Yaskawa INFORM job: A_ROOF_SIDE_0617_2_PAINT_14.JBI

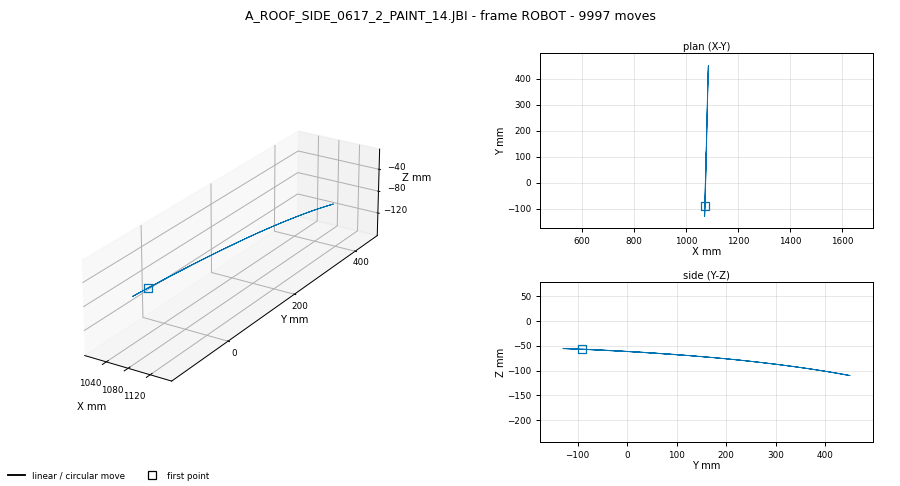
[picture p0: tool path of A_ROOF_SIDE_0617_2_PAINT_14.JBI in frame ROBOT, 9997 of 9997 moves have a stored position in this frame; points joined in program order, loops and branches not executed]
/JOB
//NAME A_ROOF_SIDE_0617_2_PAINT14
//POS
///NPOS 9997,0,0,0,0,0
///TOOL 1
///USER 0
///POSTYPE ROBOT
///RECTAN
///RCONF 1,0,0,0,0,0,0,0,0,0,0,0,0,0,0,0,0,0,0,0,0,0,0,0
C00000=1074.088,-91.546,-56.460,172.902,21.218,153.796
C00001=1074.095,-91.297,-56.470,172.904,21.219,153.796
C00002=1074.101,-91.048,-56.481,172.905,21.220,153.796
C00003=1074.107,-90.797,-56.491,172.907,21.222,153.796
C00004=1074.113,-90.548,-56.502,172.908,21.223,153.796
C00005=1074.120,-90.298,-56.512,172.910,21.225,153.796
C00006=1074.125,-90.048,-56.522,172.911,21.226,153.796
C00007=1074.131,-89.799,-56.533,172.913,21.228,153.796
C00008=1074.138,-89.549,-56.544,172.914,21.229,153.796
C00009=1074.143,-89.299,-56.554,172.916,21.231,153.796
C00010=1074.150,-89.050,-56.564,172.917,21.232,153.796
C00011=1074.156,-88.800,-56.575,172.919,21.234,153.796
C00012=1074.161,-88.550,-56.585,172.921,21.235,153.796
C00013=1074.168,-88.300,-56.596,172.922,21.237,153.796
C00014=1074.174,-88.051,-56.607,172.924,21.238,153.796
C00015=1074.180,-87.801,-56.617,172.925,21.239,153.796
C00016=1074.186,-87.551,-56.627,172.927,21.241,153.797
C00017=1074.192,-87.301,-56.639,172.928,21.242,153.797
C00018=1074.198,-87.052,-56.649,172.930,21.244,153.797
C00019=1074.204,-86.803,-56.660,172.931,21.246,153.797
C00020=1074.210,-86.552,-56.670,172.933,21.247,153.797
C00021=1074.217,-86.303,-56.681,172.934,21.248,153.797
C00022=1074.222,-86.053,-56.692,172.936,21.250,153.797
C00023=1074.229,-85.804,-56.702,172.937,21.251,153.797
C00024=1074.235,-85.554,-56.713,172.939,21.253,153.797
C00025=1074.241,-85.304,-56.723,172.941,21.254,153.797
C00026=1074.247,-85.054,-56.734,172.942,21.255,153.797
C00027=1074.253,-84.805,-56.744,172.943,21.257,153.797
C00028=1074.259,-84.555,-56.756,172.945,21.259,153.797
C00029=1074.266,-84.306,-56.766,172.947,21.260,153.797
C00030=1074.271,-84.055,-56.776,172.948,21.262,153.797
C00031=1074.277,-83.806,-56.787,172.950,21.263,153.797
C00032=1074.284,-83.556,-56.798,172.951,21.264,153.797
C00033=1074.290,-83.307,-56.808,172.953,21.266,153.797
C00034=1074.296,-83.057,-56.819,172.954,21.268,153.797
C00035=1074.303,-82.807,-56.830,172.956,21.269,153.797
C00036=1074.308,-82.558,-56.841,172.957,21.271,153.797
C00037=1074.314,-82.308,-56.851,172.959,21.272,153.797
C00038=1074.321,-82.029,-56.863,172.961,21.274,153.797
C00039=1074.328,-81.750,-56.875,172.962,21.276,153.797
C00040=1074.335,-81.471,-56.887,172.964,21.277,153.797
C00041=1074.342,-81.192,-56.899,172.965,21.279,153.798
C00042=1074.348,-80.942,-56.910,172.967,21.281,153.798
C00043=1074.354,-80.693,-56.921,172.968,21.282,153.798
C00044=1074.361,-80.443,-56.932,172.971,21.284,153.798
C00045=1074.366,-80.193,-56.943,172.972,21.285,153.798
C00046=1074.372,-79.944,-56.953,172.974,21.287,153.798
C00047=1074.379,-79.694,-56.964,172.975,21.289,153.798
C00048=1074.385,-79.444,-56.975,172.977,21.290,153.798
C00049=1074.391,-79.195,-56.986,172.978,21.292,153.798
C00050=1074.397,-78.945,-56.997,172.980,21.294,153.798
C00051=1074.403,-78.695,-57.008,172.981,21.295,153.798
C00052=1074.409,-78.446,-57.019,172.983,21.297,153.798
C00053=1074.415,-78.196,-57.030,172.984,21.298,153.798
C00054=1074.421,-77.946,-57.041,172.986,21.300,153.798
C00055=1074.426,-77.697,-57.052,172.987,21.302,153.798
C00056=1074.434,-77.447,-57.062,172.989,21.303,153.798
C00057=1074.439,-77.197,-57.073,172.990,21.305,153.799
C00058=1074.445,-76.948,-57.084,172.992,21.306,153.799
C00059=1074.451,-76.698,-57.095,172.993,21.308,153.799
C00060=1074.457,-76.448,-57.106,172.995,21.310,153.799
C00061=1074.463,-76.199,-57.117,172.996,21.311,153.799
C00062=1074.469,-75.948,-57.128,172.997,21.313,153.799
C00063=1074.475,-75.699,-57.139,172.999,21.315,153.799
C00064=1074.481,-75.449,-57.150,173.001,21.316,153.799
C00065=1074.487,-75.199,-57.161,173.002,21.318,153.799
C00066=1074.493,-74.950,-57.172,173.003,21.319,153.799
C00067=1074.500,-74.700,-57.183,173.005,21.321,153.799
C00068=1074.506,-74.450,-57.194,173.006,21.323,153.799
C00069=1074.512,-74.201,-57.205,173.008,21.324,153.799
C00070=1074.518,-73.951,-57.217,173.009,21.326,153.800
C00071=1074.524,-73.702,-57.228,173.011,21.328,153.800
C00072=1074.529,-73.452,-57.238,173.012,21.329,153.800
C00073=1074.535,-73.202,-57.250,173.014,21.331,153.800
C00074=1074.541,-72.952,-57.261,173.015,21.333,153.800
C00075=1074.547,-72.702,-57.272,173.016,21.335,153.800
C00076=1074.553,-72.453,-57.283,173.019,21.337,153.800
C00077=1074.559,-72.204,-57.295,173.020,21.339,153.800
C00078=1074.565,-71.954,-57.306,173.022,21.340,153.800
C00079=1074.571,-71.704,-57.317,173.023,21.342,153.800
C00080=1074.577,-71.455,-57.328,173.025,21.343,153.800
C00081=1074.582,-71.204,-57.340,173.026,21.345,153.800
C00082=1074.588,-70.955,-57.351,173.027,21.347,153.801
C00083=1074.594,-70.706,-57.362,173.029,21.349,153.801
C00084=1074.600,-70.456,-57.373,173.030,21.351,153.801
C00085=1074.606,-70.206,-57.384,173.032,21.352,153.801
C00086=1074.612,-69.956,-57.396,173.033,21.354,153.801
C00087=1074.619,-69.707,-57.407,173.035,21.356,153.801
C00088=1074.624,-69.457,-57.419,173.036,21.357,153.801
C00089=1074.630,-69.207,-57.430,173.037,21.359,153.801
C00090=1074.636,-68.957,-57.441,173.039,21.361,153.801
C00091=1074.642,-68.708,-57.453,173.040,21.363,153.802
C00092=1074.648,-68.458,-57.464,173.042,21.365,153.802
C00093=1074.654,-68.209,-57.474,173.043,21.366,153.802
C00094=1074.660,-67.959,-57.487,173.045,21.368,153.802
C00095=1074.665,-67.710,-57.498,173.046,21.370,153.802
C00096=1074.672,-67.459,-57.509,173.048,21.372,153.802
C00097=1074.677,-67.210,-57.520,173.050,21.374,153.802
C00098=1074.684,-66.960,-57.532,173.051,21.376,153.802
C00099=1074.690,-66.711,-57.543,173.053,21.377,153.802
C00100=1074.695,-66.460,-57.555,173.054,21.379,153.802
C00101=1074.701,-66.211,-57.566,173.055,21.381,153.803
C00102=1074.708,-65.934,-57.579,173.057,21.383,153.803
C00103=1074.715,-65.658,-57.592,173.058,21.384,153.803
C00104=1074.721,-65.381,-57.604,173.060,21.387,153.803
C00105=1074.728,-65.104,-57.616,173.062,21.389,153.803
C00106=1074.734,-64.855,-57.628,173.063,21.391,153.803
C00107=1074.740,-64.605,-57.639,173.065,21.392,153.803
C00108=1074.747,-64.356,-57.651,173.066,21.394,153.803
C00109=1074.752,-64.106,-57.662,173.067,21.396,153.804
C00110=1074.758,-63.856,-57.674,173.069,21.397,153.804
C00111=1074.764,-63.607,-57.685,173.070,21.399,153.804
C00112=1074.770,-63.357,-57.697,173.072,21.401,153.804
C00113=1074.776,-63.107,-57.709,173.073,21.403,153.804
C00114=1074.782,-62.857,-57.720,173.075,21.405,153.804
C00115=1074.788,-62.608,-57.732,173.077,21.407,153.804
C00116=1074.794,-62.358,-57.743,173.078,21.409,153.804
C00117=1074.800,-62.109,-57.754,173.080,21.410,153.804
C00118=1074.806,-61.859,-57.766,173.081,21.412,153.804
C00119=1074.812,-61.609,-57.777,173.082,21.414,153.805
C00120=1074.818,-61.360,-57.789,173.084,21.416,153.805
C00121=1074.825,-61.109,-57.800,173.085,21.418,153.805
C00122=1074.830,-60.860,-57.813,173.087,21.420,153.805
C00123=1074.836,-60.610,-57.824,173.088,21.422,153.805
C00124=1074.842,-60.361,-57.835,173.090,21.423,153.805
C00125=1074.849,-60.111,-57.847,173.091,21.425,153.805
C00126=1074.854,-59.862,-57.859,173.092,21.427,153.805
C00127=1074.860,-59.612,-57.870,173.094,21.429,153.806
C00128=1074.867,-59.362,-57.882,173.095,21.430,153.806
C00129=1074.872,-59.112,-57.893,173.097,21.433,153.806
C00130=1074.879,-58.863,-57.905,173.099,21.435,153.806
C00131=1074.884,-58.613,-57.916,173.100,21.437,153.806
C00132=1074.891,-58.364,-57.928,173.102,21.438,153.806
C00133=1074.897,-58.114,-57.941,173.103,21.440,153.806
C00134=1074.903,-57.864,-57.952,173.104,21.442,153.806
C00135=1074.909,-57.615,-57.964,173.106,21.444,153.807
C00136=1074.914,-57.365,-57.975,173.107,21.446,153.807
C00137=1074.921,-57.115,-57.987,173.109,21.447,153.807
C00138=1074.928,-56.866,-57.999,173.110,21.449,153.807
C00139=1074.933,-56.616,-58.010,173.111,21.451,153.807
C00140=1074.939,-56.366,-58.022,173.113,21.453,153.807
C00141=1074.946,-56.116,-58.034,173.114,21.455,153.807
C00142=1074.952,-55.867,-58.045,173.117,21.457,153.807
C00143=1074.958,-55.617,-58.058,173.118,21.459,153.807
C00144=1074.964,-55.367,-58.069,173.119,21.461,153.808
C00145=1074.970,-55.118,-58.081,173.121,21.463,153.808
C00146=1074.976,-54.869,-58.093,173.122,21.465,153.808
C00147=1074.982,-54.618,-58.104,173.124,21.466,153.808
C00148=1074.988,-54.369,-58.116,173.125,21.468,153.808
C00149=1074.994,-54.120,-58.129,173.126,21.470,153.808
C00150=1075.001,-53.869,-58.140,173.128,21.472,153.808
C00151=1075.007,-53.621,-58.151,173.129,21.474,153.809
C00152=1075.013,-53.371,-58.164,173.130,21.476,153.809
C00153=1075.019,-53.120,-58.175,173.132,21.477,153.809
C00154=1075.025,-52.872,-58.187,173.134,21.480,153.809
C00155=1075.031,-52.622,-58.199,173.135,21.482,153.809
C00156=1075.037,-52.372,-58.211,173.137,21.484,153.809
C00157=1075.043,-52.123,-58.222,173.138,21.486,153.809
C00158=1075.049,-51.873,-58.235,173.140,21.487,153.810
C00159=1075.056,-51.623,-58.247,173.141,21.489,153.810
C00160=1075.062,-51.374,-58.259,173.142,21.491,153.810
C00161=1075.067,-51.124,-58.270,173.144,21.493,153.810
C00162=1075.074,-50.874,-58.282,173.145,21.495,153.810
C00163=1075.080,-50.624,-58.295,173.147,21.497,153.810
C00164=1075.087,-50.375,-58.307,173.148,21.499,153.810
C00165=1075.092,-50.126,-58.319,173.150,21.501,153.810
C00166=1075.098,-49.850,-58.332,173.152,21.503,153.811
C00167=1075.105,-49.574,-58.345,173.153,21.505,153.811
C00168=1075.112,-49.299,-58.359,173.154,21.507,153.811
C00169=1075.118,-49.023,-58.372,173.156,21.510,153.811
C00170=1075.124,-48.774,-58.383,173.158,21.512,153.811
C00171=1075.130,-48.524,-58.396,173.159,21.514,153.811
C00172=1075.136,-48.274,-58.408,173.160,21.516,153.812
C00173=1075.142,-48.025,-58.420,173.162,21.518,153.812
C00174=1075.148,-47.776,-58.432,173.163,21.520,153.812
C00175=1075.154,-47.525,-58.444,173.164,21.521,153.812
C00176=1075.160,-47.276,-58.456,173.166,21.523,153.812
C00177=1075.166,-47.026,-58.468,173.168,21.526,153.812
C00178=1075.172,-46.777,-58.480,173.169,21.528,153.812
C00179=1075.178,-46.527,-58.493,173.171,21.530,153.813
C00180=1075.184,-46.278,-58.505,173.172,21.532,153.813
C00181=1075.190,-46.028,-58.517,173.173,21.534,153.813
C00182=1075.196,-45.778,-58.530,173.175,21.536,153.813
C00183=1075.201,-45.529,-58.542,173.176,21.537,153.813
C00184=1075.208,-45.279,-58.554,173.178,21.539,153.813
C00185=1075.214,-45.030,-58.566,173.179,21.542,153.814
C00186=1075.220,-44.780,-58.579,173.181,21.544,153.814
C00187=1075.226,-44.530,-58.590,173.182,21.546,153.814
C00188=1075.232,-44.280,-58.602,173.184,21.548,153.814
C00189=1075.237,-44.030,-58.615,173.185,21.550,153.814
C00190=1075.244,-43.781,-58.627,173.186,21.552,153.814
C00191=1075.249,-43.532,-58.639,173.188,21.554,153.815
C00192=1075.255,-43.282,-58.652,173.189,21.556,153.815
C00193=1075.262,-43.032,-58.664,173.190,21.558,153.815
C00194=1075.268,-42.782,-58.676,173.192,21.560,153.815
C00195=1075.273,-42.533,-58.688,173.193,21.562,153.815
C00196=1075.279,-42.283,-58.701,173.195,21.565,153.815
C00197=1075.286,-42.034,-58.713,173.197,21.567,153.816
C00198=1075.292,-41.784,-58.725,173.198,21.569,153.816
C00199=1075.298,-41.535,-58.739,173.199,21.571,153.816
C00200=1075.304,-41.286,-58.750,173.201,21.573,153.816
C00201=1075.310,-41.036,-58.763,173.202,21.574,153.816
C00202=1075.316,-40.786,-58.775,173.203,21.576,153.816
C00203=1075.322,-40.536,-58.788,173.205,21.578,153.817
C00204=1075.328,-40.286,-58.800,173.206,21.580,153.817
C00205=1075.334,-40.037,-58.812,173.208,21.583,153.817
C00206=1075.340,-39.787,-58.825,173.209,21.585,153.817
C00207=1075.346,-39.538,-58.837,173.211,21.587,153.817
C00208=1075.352,-39.288,-58.849,173.212,21.589,153.817
C00209=1075.358,-39.038,-58.862,173.214,21.591,153.818
C00210=1075.364,-38.789,-58.875,173.215,21.593,153.818
C00211=1075.371,-38.539,-58.887,173.216,21.595,153.818
C00212=1075.376,-38.290,-58.899,173.217,21.597,153.818
C00213=1075.382,-38.040,-58.912,173.219,21.599,153.818
C00214=1075.388,-37.790,-58.924,173.221,21.602,153.818
C00215=1075.394,-37.540,-58.937,173.222,21.604,153.819
C00216=1075.400,-37.291,-58.949,173.224,21.606,153.819
C00217=1075.405,-37.042,-58.962,173.225,21.608,153.819
C00218=1075.411,-36.792,-58.975,173.226,21.610,153.819
C00219=1075.417,-36.542,-58.987,173.228,21.612,153.819
C00220=1075.423,-36.292,-59.000,173.229,21.614,153.820
C00221=1075.429,-36.042,-59.012,173.230,21.616,153.820
C00222=1075.435,-35.794,-59.025,173.232,21.619,153.820
C00223=1075.441,-35.544,-59.037,173.234,21.621,153.820
C00224=1075.447,-35.294,-59.050,173.235,21.623,153.820
C00225=1075.453,-35.045,-59.062,173.236,21.625,153.821
C00226=1075.459,-34.795,-59.075,173.238,21.627,153.821
C00227=1075.465,-34.545,-59.088,173.239,21.629,153.821
C00228=1075.471,-34.295,-59.101,173.240,21.632,153.821
C00229=1075.476,-34.046,-59.113,173.242,21.633,153.821
C00230=1075.484,-33.772,-59.127,173.244,21.636,153.821
C00231=1075.490,-33.496,-59.141,173.245,21.638,153.822
C00232=1075.497,-33.221,-59.156,173.246,21.640,153.822
C00233=1075.503,-32.946,-59.169,173.248,21.643,153.822
C00234=1075.509,-32.696,-59.182,173.250,21.645,153.822
C00235=1075.515,-32.447,-59.195,173.251,21.648,153.823
C00236=1075.521,-32.198,-59.207,173.252,21.650,153.823
C00237=1075.527,-31.948,-59.220,173.254,21.651,153.823
C00238=1075.533,-31.698,-59.233,173.255,21.653,153.823
C00239=1075.539,-31.449,-59.246,173.257,21.656,153.823
C00240=1075.545,-31.199,-59.258,173.258,21.658,153.823
C00241=1075.551,-30.949,-59.271,173.260,21.660,153.824
C00242=1075.557,-30.699,-59.284,173.261,21.663,153.824
C00243=1075.563,-30.450,-59.297,173.262,21.665,153.824
C00244=1075.569,-30.200,-59.310,173.264,21.667,153.824
C00245=1075.575,-29.950,-59.322,173.265,21.669,153.825
C00246=1075.581,-29.701,-59.335,173.266,21.671,153.825
C00247=1075.587,-29.451,-59.348,173.269,21.673,153.825
C00248=1075.593,-29.201,-59.361,173.270,21.675,153.825
C00249=1075.599,-28.952,-59.374,173.271,21.678,153.825
C00250=1075.605,-28.702,-59.387,173.272,21.680,153.825
C00251=1075.611,-28.453,-59.400,173.274,21.682,153.826
C00252=1075.617,-28.204,-59.412,173.275,21.684,153.826
C00253=1075.622,-27.954,-59.425,173.276,21.686,153.826
C00254=1075.629,-27.705,-59.438,173.278,21.688,153.826
C00255=1075.635,-27.455,-59.450,173.280,21.691,153.826
C00256=1075.641,-27.206,-59.464,173.281,21.693,153.827
C00257=1075.647,-26.956,-59.476,173.282,21.695,153.827
C00258=1075.653,-26.706,-59.489,173.284,21.697,153.827
C00259=1075.658,-26.456,-59.503,173.285,21.699,153.827
C00260=1075.664,-26.207,-59.516,173.286,21.702,153.827
C00261=1075.670,-25.957,-59.528,173.288,21.704,153.828
C00262=1075.676,-25.708,-59.542,173.290,21.706,153.828
C00263=1075.682,-25.458,-59.554,173.291,21.709,153.828
C00264=1075.688,-25.208,-59.568,173.292,21.710,153.828
C00265=1075.694,-24.958,-59.581,173.294,21.713,153.828
C00266=1075.700,-24.709,-59.594,173.295,21.715,153.829
C00267=1075.706,-24.459,-59.607,173.296,21.717,153.829
C00268=1075.712,-24.210,-59.620,173.297,21.719,153.829
C00269=1075.718,-23.960,-59.634,173.300,21.722,153.829
C00270=1075.723,-23.711,-59.646,173.301,21.724,153.830
C00271=1075.730,-23.461,-59.659,173.302,21.726,153.830
C00272=1075.736,-23.211,-59.672,173.303,21.729,153.830
C00273=1075.741,-22.962,-59.686,173.305,21.730,153.830
C00274=1075.747,-22.712,-59.698,173.306,21.733,153.830
C00275=1075.753,-22.463,-59.712,173.307,21.735,153.831
C00276=1075.759,-22.213,-59.725,173.308,21.737,153.831
C00277=1075.765,-21.963,-59.738,173.311,21.740,153.831
C00278=1075.771,-21.714,-59.751,173.312,21.742,153.831
C00279=1075.777,-21.465,-59.765,173.313,21.744,153.831
C00280=1075.783,-21.215,-59.777,173.315,21.746,153.832
C00281=1075.788,-20.965,-59.791,173.316,21.749,153.832
C00282=1075.795,-20.716,-59.804,173.317,21.751,153.832
C00283=1075.800,-20.466,-59.817,173.318,21.753,153.832
C00284=1075.807,-20.217,-59.830,173.321,21.755,153.832
C00285=1075.812,-19.967,-59.844,173.322,21.758,153.833
C00286=1075.818,-19.717,-59.857,173.323,21.760,153.833
C00287=1075.824,-19.468,-59.870,173.324,21.762,153.833
C00288=1075.831,-19.219,-59.883,173.326,21.764,153.833
C00289=1075.836,-18.969,-59.896,173.327,21.767,153.834
C00290=1075.842,-18.719,-59.910,173.328,21.769,153.834
C00291=1075.849,-18.469,-59.923,173.330,21.772,153.834
C00292=1075.854,-18.220,-59.937,173.332,21.773,153.834
C00293=1075.860,-17.970,-59.950,173.333,21.776,153.834
C00294=1075.866,-17.695,-59.964,173.334,21.778,153.835
C00295=1075.873,-17.419,-59.979,173.336,21.781,153.835
C00296=1075.880,-17.143,-59.994,173.337,21.783,153.835
C00297=1075.887,-16.866,-60.009,173.339,21.785,153.835
C00298=1075.893,-16.617,-60.022,173.341,21.788,153.836
C00299=1075.899,-16.368,-60.035,173.342,21.790,153.836
C00300=1075.904,-16.118,-60.048,173.343,21.792,153.836
C00301=1075.910,-15.868,-60.062,173.345,21.794,153.836
C00302=1075.917,-15.619,-60.075,173.346,21.797,153.836
C00303=1075.922,-15.370,-60.089,173.347,21.799,153.837
C00304=1075.928,-15.120,-60.102,173.349,21.801,153.837
C00305=1075.935,-14.870,-60.116,173.351,21.804,153.837
C00306=1075.940,-14.620,-60.129,173.352,21.806,153.837
C00307=1075.947,-14.371,-60.142,173.353,21.809,153.838
C00308=1075.952,-14.121,-60.156,173.354,21.811,153.838
C00309=1075.958,-13.872,-60.169,173.356,21.813,153.838
C00310=1075.964,-13.623,-60.183,173.357,21.815,153.838
C00311=1075.970,-13.373,-60.196,173.359,21.818,153.839
C00312=1075.975,-13.124,-60.210,173.360,21.820,153.839
C00313=1075.981,-12.874,-60.223,173.362,21.822,153.839
C00314=1075.987,-12.624,-60.237,173.363,21.825,153.839
C00315=1075.994,-12.374,-60.250,173.364,21.827,153.839
C00316=1075.999,-12.125,-60.264,173.365,21.829,153.840
C00317=1076.005,-11.875,-60.277,173.367,21.831,153.840
C00318=1076.011,-11.626,-60.291,173.369,21.834,153.840
C00319=1076.016,-11.376,-60.305,173.370,21.836,153.840
C00320=1076.022,-11.127,-60.318,173.371,21.838,153.841
C00321=1076.028,-10.877,-60.332,173.373,21.841,153.841
C00322=1076.035,-10.627,-60.346,173.374,21.843,153.841
C00323=1076.040,-10.378,-60.360,173.375,21.845,153.841
C00324=1076.046,-10.129,-60.373,173.377,21.848,153.842
C00325=1076.052,-9.879,-60.387,173.379,21.850,153.842
C00326=1076.058,-9.630,-60.400,173.380,21.853,153.842
C00327=1076.064,-9.380,-60.414,173.381,21.855,153.842
C00328=1076.070,-9.130,-60.428,173.382,21.857,153.842
C00329=1076.076,-8.881,-60.442,173.383,21.859,153.843
C00330=1076.082,-8.631,-60.455,173.386,21.862,153.843
C00331=1076.088,-8.382,-60.469,173.387,21.864,153.843
C00332=1076.093,-8.132,-60.483,173.388,21.866,153.843
C00333=1076.100,-7.882,-60.496,173.389,21.869,153.844
C00334=1076.105,-7.633,-60.510,173.391,21.871,153.844
C00335=1076.112,-7.383,-60.523,173.392,21.873,153.844
C00336=1076.117,-7.134,-60.537,173.393,21.876,153.844
C00337=1076.123,-6.885,-60.550,173.395,21.878,153.844
C00338=1076.129,-6.634,-60.565,173.397,21.880,153.845
C00339=1076.135,-6.385,-60.579,173.398,21.883,153.845
C00340=1076.141,-6.135,-60.592,173.399,21.885,153.845
C00341=1076.147,-5.887,-60.606,173.400,21.887,153.846
C00342=1076.154,-5.637,-60.620,173.402,21.889,153.846
C00343=1076.159,-5.387,-60.634,173.404,21.892,153.846
C00344=1076.165,-5.137,-60.648,173.405,21.895,153.846
C00345=1076.171,-4.888,-60.661,173.406,21.896,153.846
C00346=1076.177,-4.638,-60.675,173.408,21.899,153.847
C00347=1076.183,-4.389,-60.689,173.409,21.901,153.847
C00348=1076.189,-4.139,-60.702,173.410,21.903,153.847
C00349=1076.195,-3.889,-60.717,173.412,21.906,153.847
C00350=1076.201,-3.640,-60.731,173.414,21.908,153.848
C00351=1076.207,-3.391,-60.745,173.415,21.911,153.848
C00352=1076.212,-3.141,-60.758,173.416,21.913,153.848
C00353=1076.219,-2.891,-60.772,173.417,21.915,153.848
C00354=1076.225,-2.642,-60.787,173.419,21.918,153.849
C00355=1076.230,-2.392,-60.800,173.421,21.920,153.849
C00356=1076.236,-2.143,-60.814,173.422,21.923,153.849
C00357=1076.241,-1.893,-60.828,173.423,21.925,153.849
C00358=1076.248,-1.616,-60.844,173.424,21.927,153.850
C00359=1076.255,-1.338,-60.859,173.426,21.930,153.850
C00360=1076.261,-1.060,-60.875,173.428,21.933,153.850
C00361=1076.268,-0.783,-60.890,173.429,21.936,153.850
C00362=1076.273,-0.534,-60.905,173.431,21.938,153.851
C00363=1076.279,-0.284,-60.919,173.432,21.940,153.851
C00364=1076.285,-0.034,-60.933,173.433,21.943,153.851
C00365=1076.290,0.215,-60.947,173.434,21.945,153.852
C00366=1076.296,0.464,-60.962,173.436,21.947,153.852
C00367=1076.302,0.714,-60.975,173.438,21.950,153.852
C00368=1076.309,0.964,-60.989,173.439,21.953,153.852
C00369=1076.314,1.213,-61.004,173.440,21.955,153.853
C00370=1076.320,1.462,-61.018,173.442,21.957,153.853
C00371=1076.325,1.712,-61.031,173.443,21.960,153.853
C00372=1076.332,1.962,-61.046,173.444,21.962,153.853
C00373=1076.337,2.211,-61.060,173.446,21.964,153.853
C00374=1076.343,2.461,-61.074,173.447,21.967,153.854
C00375=1076.349,2.710,-61.089,173.449,21.969,153.854
C00376=1076.355,2.960,-61.102,173.450,21.972,153.854
C00377=1076.361,3.209,-61.116,173.451,21.974,153.854
C00378=1076.367,3.459,-61.131,173.452,21.976,153.855
C00379=1076.373,3.709,-61.145,173.454,21.979,153.855
C00380=1076.378,3.957,-61.160,173.456,21.981,153.855
C00381=1076.384,4.208,-61.174,173.457,21.983,153.855
C00382=1076.390,4.457,-61.188,173.458,21.986,153.856
C00383=1076.396,4.706,-61.202,173.459,21.988,153.856
C00384=1076.402,4.957,-61.216,173.461,21.991,153.856
C00385=1076.408,5.206,-61.231,173.463,21.993,153.856
C00386=1076.413,5.455,-61.245,173.464,21.996,153.857
C00387=1076.419,5.705,-61.260,173.465,21.998,153.857
C00388=1076.425,5.954,-61.274,173.466,22.001,153.857
C00389=1076.431,6.203,-61.288,173.468,22.002,153.857
C00390=1076.437,6.453,-61.302,173.470,22.005,153.858
C00391=1076.443,6.702,-61.316,173.471,22.008,153.858
C00392=1076.449,6.952,-61.331,173.472,22.010,153.858
C00393=1076.455,7.201,-61.345,173.474,22.012,153.858
C00394=1076.461,7.451,-61.359,173.475,22.015,153.859
C00395=1076.467,7.701,-61.374,173.476,22.017,153.859
C00396=1076.472,7.950,-61.388,173.478,22.020,153.859
C00397=1076.479,8.200,-61.403,173.480,22.022,153.859
C00398=1076.484,8.449,-61.417,173.481,22.024,153.860
C00399=1076.490,8.698,-61.431,173.482,22.027,153.860
C00400=1076.496,8.949,-61.446,173.483,22.029,153.860
C00401=1076.502,9.198,-61.460,173.485,22.032,153.860
C00402=1076.508,9.448,-61.474,173.487,22.034,153.861
C00403=1076.514,9.697,-61.489,173.488,22.037,153.861
C00404=1076.520,9.947,-61.504,173.489,22.039,153.861
C00405=1076.526,10.196,-61.518,173.490,22.041,153.862
C00406=1076.532,10.446,-61.533,173.492,22.043,153.862
C00407=1076.537,10.695,-61.547,173.494,22.046,153.862
C00408=1076.543,10.944,-61.561,173.495,22.048,153.862
C00409=1076.550,11.194,-61.576,173.496,22.051,153.862
C00410=1076.555,11.444,-61.590,173.497,22.053,153.863
C00411=1076.562,11.693,-61.605,173.499,22.056,153.863
C00412=1076.567,11.942,-61.620,173.501,22.058,153.863
C00413=1076.573,12.192,-61.634,173.502,22.060,153.863
C00414=1076.579,12.441,-61.648,173.503,22.063,153.864
C00415=1076.586,12.691,-61.663,173.505,22.065,153.864
C00416=1076.591,12.941,-61.677,173.506,22.067,153.864
C00417=1076.597,13.190,-61.692,173.508,22.070,153.864
C00418=1076.603,13.439,-61.707,173.509,22.073,153.865
C00419=1076.609,13.690,-61.721,173.510,22.075,153.865
C00420=1076.615,13.938,-61.735,173.512,22.077,153.865
C00421=1076.621,14.188,-61.750,173.513,22.079,153.866
C00422=1076.628,14.468,-61.766,173.515,22.082,153.866
C00423=1076.635,14.747,-61.783,173.516,22.085,153.866
C00424=1076.641,15.026,-61.799,173.518,22.088,153.866
C00425=1076.647,15.306,-61.816,173.519,22.090,153.867
C00426=1076.653,15.556,-61.831,173.521,22.093,153.867
C00427=1076.659,15.805,-61.845,173.522,22.095,153.867
C00428=1076.665,16.054,-61.860,173.524,22.098,153.867
C00429=1076.671,16.304,-61.875,173.525,22.100,153.868
C00430=1076.677,16.554,-61.890,173.526,22.102,153.868
C00431=1076.682,16.803,-61.904,173.528,22.105,153.868
C00432=1076.689,17.053,-61.919,173.529,22.107,153.869
C00433=1076.695,17.302,-61.934,173.531,22.110,153.869
C00434=1076.700,17.552,-61.949,173.532,22.113,153.869
C00435=1076.706,17.801,-61.963,173.534,22.114,153.869
C00436=1076.712,18.051,-61.978,173.535,22.117,153.870
C00437=1076.718,18.300,-61.993,173.536,22.119,153.870
C00438=1076.723,18.550,-62.008,173.538,22.122,153.870
C00439=1076.729,18.799,-62.023,173.539,22.125,153.870
C00440=1076.736,19.048,-62.038,173.540,22.127,153.871
C00441=1076.741,19.297,-62.052,173.542,22.129,153.871
C00442=1076.747,19.548,-62.067,173.543,22.132,153.871
C00443=1076.753,19.797,-62.082,173.545,22.134,153.871
C00444=1076.759,20.046,-62.097,173.546,22.137,153.872
C00445=1076.765,20.296,-62.112,173.548,22.139,153.872
C00446=1076.770,20.545,-62.127,173.549,22.141,153.872
C00447=1076.777,20.795,-62.142,173.550,22.144,153.872
C00448=1076.783,21.044,-62.156,173.552,22.147,153.873
C00449=1076.788,21.294,-62.172,173.553,22.149,153.873
C00450=1076.794,21.543,-62.186,173.555,22.151,153.873
C00451=1076.800,21.793,-62.202,173.556,22.154,153.874
C00452=1076.805,22.042,-62.216,173.557,22.156,153.874
C00453=1076.812,22.291,-62.231,173.559,22.159,153.874
C00454=1076.817,22.541,-62.247,173.560,22.161,153.874
C00455=1076.823,22.790,-62.262,173.562,22.164,153.875
C00456=1076.830,23.040,-62.277,173.563,22.166,153.875
C00457=1076.835,23.289,-62.292,173.564,22.169,153.875
C00458=1076.841,23.539,-62.307,173.566,22.171,153.875
C00459=1076.847,23.789,-62.322,173.568,22.173,153.876
C00460=1076.852,24.038,-62.337,173.569,22.176,153.876
C00461=1076.859,24.288,-62.352,173.570,22.178,153.876
C00462=1076.864,24.537,-62.367,173.571,22.181,153.876
C00463=1076.870,24.786,-62.382,173.573,22.184,153.877
C00464=1076.876,25.036,-62.397,173.574,22.186,153.877
C00465=1076.882,25.285,-62.412,173.576,22.188,153.877
C00466=1076.888,25.535,-62.427,173.577,22.190,153.877
C00467=1076.893,25.784,-62.442,173.578,22.193,153.878
C00468=1076.899,26.034,-62.457,173.580,22.196,153.878
C00469=1076.905,26.284,-62.473,173.582,22.198,153.878
C00470=1076.911,26.533,-62.487,173.583,22.200,153.878
C00471=1076.917,26.783,-62.502,173.584,22.202,153.879
C00472=1076.923,27.032,-62.518,173.585,22.205,153.879
C00473=1076.929,27.281,-62.533,173.587,22.208,153.879
C00474=1076.935,27.531,-62.548,173.589,22.210,153.880
C00475=1076.940,27.780,-62.563,173.590,22.213,153.880
C00476=1076.946,28.030,-62.579,173.591,22.215,153.880
C00477=1076.952,28.279,-62.594,173.593,22.218,153.880
C00478=1076.958,28.529,-62.609,173.595,22.220,153.881
C00479=1076.964,28.778,-62.624,173.596,22.222,153.881
C00480=1076.970,29.028,-62.640,173.597,22.225,153.881
C00481=1076.976,29.277,-62.654,173.598,22.227,153.881
C00482=1076.981,29.527,-62.670,173.600,22.230,153.882
C00483=1076.987,29.777,-62.686,173.601,22.233,153.882
C00484=1076.993,30.025,-62.701,173.603,22.235,153.882
C00485=1076.999,30.275,-62.716,173.604,22.237,153.882
C00486=1077.005,30.556,-62.733,173.606,22.240,153.883
C00487=1077.012,30.836,-62.750,173.607,22.243,153.883
C00488=1077.018,31.117,-62.768,173.609,22.246,153.883
C00489=1077.025,31.399,-62.785,173.611,22.248,153.884
C00490=1077.031,31.647,-62.801,173.612,22.251,153.884
C00491=1077.036,31.897,-62.816,173.614,22.253,153.884
C00492=1077.043,32.147,-62.831,173.615,22.256,153.885
C00493=1077.048,32.396,-62.847,173.616,22.258,153.885
C00494=1077.054,32.624,-62.861,173.618,22.260,153.885
C00495=1077.059,32.853,-62.875,173.619,22.263,153.885
C00496=1077.064,33.081,-62.890,173.620,22.265,153.886
C00497=1077.069,33.310,-62.903,173.621,22.267,153.886
C00498=1077.074,33.539,-62.917,173.623,22.270,153.886
C00499=1077.080,33.767,-62.931,173.624,22.272,153.886
C00500=1077.085,33.995,-62.946,173.625,22.274,153.886
C00501=1077.090,34.224,-62.960,173.626,22.276,153.887
C00502=1077.097,34.473,-62.975,173.629,22.279,153.887
C00503=1077.103,34.723,-62.991,173.630,22.281,153.887
C00504=1077.108,34.973,-63.007,173.631,22.284,153.888
C00505=1077.114,35.222,-63.022,173.632,22.286,153.888
C00506=1077.120,35.471,-63.038,173.634,22.289,153.888
C00507=1077.126,35.721,-63.053,173.636,22.291,153.888
C00508=1077.132,35.971,-63.068,173.637,22.294,153.889
C00509=1077.138,36.219,-63.084,173.638,22.296,153.889
C00510=1077.143,36.469,-63.100,173.640,22.298,153.889
C00511=1077.150,36.718,-63.115,173.642,22.301,153.889
C00512=1077.156,36.968,-63.131,173.643,22.303,153.890
C00513=1077.161,37.217,-63.146,173.644,22.306,153.890
C00514=1077.167,37.466,-63.162,173.645,22.308,153.890
C00515=1077.173,37.716,-63.177,173.647,22.311,153.890
C00516=1077.179,37.966,-63.194,173.649,22.313,153.891
C00517=1077.184,38.215,-63.209,173.650,22.316,153.891
C00518=1077.191,38.464,-63.224,173.651,22.318,153.891
C00519=1077.196,38.714,-63.240,173.653,22.321,153.891
C00520=1077.202,38.963,-63.256,173.654,22.323,153.892
C00521=1077.207,39.213,-63.271,173.656,22.326,153.892
C00522=1077.213,39.462,-63.288,173.657,22.328,153.892
C00523=1077.219,39.712,-63.303,173.658,22.331,153.893
C00524=1077.226,39.961,-63.319,173.660,22.333,153.893
C00525=1077.231,40.211,-63.334,173.661,22.336,153.893
C00526=1077.237,40.460,-63.350,173.663,22.338,153.893
C00527=1077.242,40.710,-63.366,173.664,22.340,153.894
C00528=1077.248,40.959,-63.382,173.666,22.343,153.894
C00529=1077.254,41.208,-63.398,173.667,22.346,153.894
C00530=1077.260,41.458,-63.414,173.669,22.348,153.895
C00531=1077.265,41.707,-63.430,173.670,22.350,153.895
C00532=1077.271,41.957,-63.445,173.672,22.353,153.895
C00533=1077.277,42.206,-63.461,173.673,22.356,153.895
C00534=1077.283,42.456,-63.477,173.675,22.358,153.896
C00535=1077.289,42.705,-63.493,173.676,22.360,153.896
C00536=1077.294,42.954,-63.509,173.678,22.363,153.896
C00537=1077.300,43.204,-63.524,173.679,22.365,153.896
C00538=1077.306,43.453,-63.541,173.680,22.368,153.897
C00539=1077.312,43.703,-63.557,173.682,22.370,153.897
C00540=1077.318,43.953,-63.572,173.684,22.373,153.897
C00541=1077.323,44.202,-63.589,173.685,22.376,153.898
C00542=1077.329,44.451,-63.604,173.686,22.378,153.898
C00543=1077.334,44.701,-63.620,173.687,22.380,153.898
C00544=1077.340,44.950,-63.636,173.689,22.383,153.898
C00545=1077.346,45.199,-63.653,173.691,22.386,153.899
C00546=1077.351,45.448,-63.668,173.692,22.388,153.899
C00547=1077.357,45.698,-63.684,173.693,22.390,153.899
C00548=1077.363,45.947,-63.700,173.695,22.393,153.899
C00549=1077.369,46.197,-63.716,173.697,22.395,153.900
C00550=1077.376,46.520,-63.737,173.698,22.399,153.900
C00551=1077.384,46.843,-63.758,173.700,22.402,153.900
C00552=1077.391,47.165,-63.778,173.702,22.406,153.901
C00553=1077.398,47.488,-63.800,173.703,22.409,153.901
C00554=1077.404,47.737,-63.816,173.706,22.411,153.901
C00555=1077.410,47.987,-63.831,173.707,22.413,153.902
C00556=1077.416,48.237,-63.848,173.708,22.416,153.902
C00557=1077.422,48.486,-63.864,173.709,22.418,153.902
C00558=1077.428,48.735,-63.880,173.711,22.421,153.903
C00559=1077.433,48.984,-63.896,173.713,22.423,153.903
C00560=1077.438,49.234,-63.912,173.714,22.426,153.903
C00561=1077.444,49.484,-63.929,173.715,22.428,153.903
C00562=1077.450,49.733,-63.945,173.717,22.431,153.904
C00563=1077.456,49.982,-63.961,173.718,22.434,153.904
C00564=1077.462,50.232,-63.977,173.720,22.436,153.904
C00565=1077.468,50.481,-63.994,173.721,22.438,153.905
C00566=1077.473,50.731,-64.009,173.723,22.441,153.905
C00567=1077.478,50.981,-64.026,173.724,22.443,153.905
C00568=1077.484,51.230,-64.042,173.726,22.446,153.905
C00569=1077.490,51.479,-64.058,173.728,22.448,153.906
C00570=1077.496,51.728,-64.074,173.729,22.451,153.906
C00571=1077.502,51.977,-64.091,173.730,22.453,153.906
C00572=1077.508,52.227,-64.107,173.731,22.456,153.906
C00573=1077.514,52.476,-64.123,173.733,22.459,153.907
C00574=1077.519,52.726,-64.140,173.735,22.461,153.907
C00575=1077.525,52.975,-64.156,173.736,22.463,153.907
C00576=1077.531,53.224,-64.173,173.737,22.465,153.907
C00577=1077.537,53.474,-64.189,173.739,22.468,153.908
C00578=1077.543,53.723,-64.205,173.741,22.471,153.908
C00579=1077.547,53.973,-64.221,173.742,22.473,153.908
C00580=1077.553,54.223,-64.237,173.743,22.476,153.909
C00581=1077.559,54.472,-64.254,173.745,22.478,153.909
C00582=1077.565,54.721,-64.270,173.747,22.480,153.909
C00583=1077.571,54.971,-64.286,173.748,22.483,153.909
C00584=1077.577,55.220,-64.302,173.750,22.486,153.910
C00585=1077.583,55.469,-64.320,173.751,22.488,153.910
C00586=1077.589,55.719,-64.336,173.752,22.490,153.910
C00587=1077.595,55.968,-64.353,173.754,22.493,153.910
C00588=1077.601,56.217,-64.369,173.756,22.495,153.911
C00589=1077.606,56.467,-64.386,173.757,22.498,153.911
C00590=1077.612,56.716,-64.402,173.758,22.500,153.911
C00591=1077.618,56.966,-64.418,173.760,22.503,153.911
C00592=1077.624,57.215,-64.434,173.762,22.505,153.912
C00593=1077.630,57.464,-64.451,173.763,22.508,153.912
C00594=1077.635,57.714,-64.467,173.764,22.510,153.912
C00595=1077.641,57.963,-64.484,173.767,22.513,153.912
C00596=1077.647,58.213,-64.500,173.768,22.515,153.913
C00597=1077.653,58.462,-64.516,173.769,22.517,153.913
C00598=1077.658,58.711,-64.534,173.770,22.520,153.913
C00599=1077.664,58.960,-64.550,173.773,22.522,153.913
C00600=1077.670,59.210,-64.566,173.774,22.525,153.914
C00601=1077.676,59.459,-64.583,173.775,22.527,153.914
C00602=1077.681,59.709,-64.599,173.776,22.529,153.914
C00603=1077.688,59.959,-64.616,173.778,22.532,153.915
C00604=1077.694,60.208,-64.633,173.780,22.534,153.915
C00605=1077.700,60.457,-64.649,173.781,22.537,153.915
C00606=1077.705,60.707,-64.666,173.783,22.539,153.915
C00607=1077.711,60.956,-64.682,173.784,22.542,153.916
C00608=1077.717,61.205,-64.699,173.786,22.544,153.916
C00609=1077.723,61.454,-64.716,173.787,22.546,153.916
C00610=1077.729,61.704,-64.732,173.789,22.549,153.916
C00611=1077.735,61.953,-64.749,173.790,22.551,153.917
C00612=1077.741,62.203,-64.765,173.792,22.554,153.917
C00613=1077.746,62.453,-64.782,173.794,22.556,153.917
C00614=1077.753,62.732,-64.801,173.795,22.559,153.917
C00615=1077.760,63.013,-64.819,173.797,22.561,153.918
C00616=1077.766,63.293,-64.839,173.798,22.564,153.918
C00617=1077.773,63.574,-64.857,173.800,22.567,153.918
C00618=1077.779,63.824,-64.873,173.802,22.569,153.918
C00619=1077.785,64.073,-64.891,173.803,22.572,153.919
C00620=1077.791,64.323,-64.908,173.805,22.574,153.919
C00621=1077.797,64.572,-64.924,173.806,22.577,153.919
C00622=1077.803,64.821,-64.941,173.808,22.579,153.919
C00623=1077.809,65.071,-64.958,173.810,22.582,153.920
C00624=1077.814,65.320,-64.975,173.811,22.584,153.920
C00625=1077.820,65.569,-64.992,173.812,22.586,153.920
C00626=1077.825,65.819,-65.008,173.814,22.589,153.921
C00627=1077.831,66.068,-65.025,173.816,22.592,153.921
C00628=1077.837,66.318,-65.043,173.817,22.594,153.921
C00629=1077.843,66.567,-65.059,173.818,22.596,153.921
C00630=1077.848,66.817,-65.076,173.820,22.599,153.922
C00631=1077.855,67.066,-65.093,173.822,22.601,153.922
C00632=1077.860,67.315,-65.110,173.823,22.604,153.922
C00633=1077.866,67.564,-65.127,173.825,22.606,153.922
C00634=1077.871,67.814,-65.143,173.826,22.608,153.923
C00635=1077.878,68.063,-65.161,173.828,22.611,153.923
C00636=1077.883,68.313,-65.178,173.830,22.614,153.923
C00637=1077.889,68.562,-65.194,173.831,22.616,153.923
C00638=1077.895,68.811,-65.211,173.833,22.618,153.924
C00639=1077.900,69.061,-65.228,173.834,22.620,153.924
C00640=1077.906,69.309,-65.245,173.836,22.623,153.924
C00641=1077.912,69.560,-65.262,173.837,22.626,153.924
C00642=1077.918,69.809,-65.280,173.838,22.628,153.925
C00643=1077.924,70.058,-65.296,173.841,22.630,153.925
C00644=1077.929,70.307,-65.314,173.842,22.633,153.925
C00645=1077.935,70.557,-65.330,173.843,22.635,153.925
C00646=1077.941,70.806,-65.348,173.845,22.638,153.926
C00647=1077.946,71.056,-65.365,173.846,22.641,153.926
C00648=1077.953,71.305,-65.382,173.848,22.643,153.926
C00649=1077.958,71.554,-65.399,173.850,22.645,153.926
C00650=1077.963,71.803,-65.416,173.851,22.648,153.927
C00651=1077.970,72.052,-65.433,173.853,22.650,153.927
C00652=1077.976,72.302,-65.450,173.854,22.653,153.927
C00653=1077.981,72.552,-65.468,173.856,22.655,153.928
C00654=1077.986,72.801,-65.485,173.857,22.657,153.928
C00655=1077.993,73.050,-65.502,173.859,22.660,153.928
C00656=1077.998,73.299,-65.519,173.861,22.662,153.928
C00657=1078.004,73.549,-65.537,173.862,22.665,153.929
C00658=1078.010,73.798,-65.554,173.863,22.667,153.929
C00659=1078.016,74.047,-65.571,173.865,22.670,153.929
C00660=1078.021,74.297,-65.588,173.867,22.672,153.929
C00661=1078.027,74.546,-65.606,173.868,22.674,153.930
C00662=1078.033,74.795,-65.623,173.870,22.677,153.930
C00663=1078.038,75.045,-65.640,173.871,22.679,153.930
C00664=1078.044,75.294,-65.657,173.873,22.682,153.930
C00665=1078.050,75.544,-65.675,173.875,22.684,153.931
C00666=1078.056,75.793,-65.692,173.876,22.687,153.931
C00667=1078.062,76.042,-65.709,173.877,22.689,153.931
C00668=1078.067,76.291,-65.727,173.880,22.692,153.931
C00669=1078.073,76.541,-65.744,173.881,22.694,153.932
C00670=1078.079,76.790,-65.761,173.882,22.696,153.932
C00671=1078.085,77.039,-65.778,173.884,22.699,153.932
C00672=1078.090,77.288,-65.796,173.886,22.701,153.932
C00673=1078.096,77.539,-65.813,173.887,22.704,153.933
C00674=1078.102,77.788,-65.831,173.889,22.706,153.933
C00675=1078.108,78.036,-65.848,173.890,22.709,153.933
C00676=1078.114,78.286,-65.866,173.892,22.711,153.933
C00677=1078.119,78.536,-65.883,173.894,22.714,153.934
C00678=1078.125,78.817,-65.903,173.895,22.716,153.934
C00679=1078.132,79.097,-65.922,173.897,22.719,153.934
C00680=1078.138,79.377,-65.942,173.898,22.721,153.934
C00681=1078.145,79.658,-65.961,173.900,22.725,153.935
C00682=1078.150,79.907,-65.979,173.902,22.726,153.935
C00683=1078.156,80.156,-65.996,173.904,22.729,153.935
C00684=1078.162,80.406,-66.014,173.905,22.732,153.936
C00685=1078.168,80.655,-66.032,173.906,22.734,153.936
C00686=1078.173,80.904,-66.049,173.909,22.737,153.936
C00687=1078.179,81.154,-66.067,173.910,22.739,153.936
C00688=1078.184,81.403,-66.084,173.911,22.741,153.937
C00689=1078.190,81.652,-66.102,173.913,22.744,153.937
C00690=1078.195,81.901,-66.119,173.915,22.746,153.937
C00691=1078.202,82.151,-66.137,173.916,22.749,153.937
C00692=1078.207,82.400,-66.155,173.918,22.751,153.938
C00693=1078.213,82.649,-66.172,173.919,22.754,153.938
C00694=1078.219,82.899,-66.190,173.922,22.756,153.938
C00695=1078.224,83.148,-66.208,173.923,22.759,153.938
C00696=1078.230,83.397,-66.225,173.924,22.761,153.939
C00697=1078.236,83.647,-66.243,173.926,22.764,153.939
C00698=1078.241,83.896,-66.261,173.928,22.766,153.939
C00699=1078.247,84.145,-66.278,173.929,22.768,153.939
C00700=1078.253,84.395,-66.296,173.931,22.771,153.940
C00701=1078.259,84.644,-66.314,173.932,22.773,153.940
C00702=1078.265,84.893,-66.332,173.934,22.775,153.940
C00703=1078.270,85.142,-66.349,173.936,22.778,153.940
C00704=1078.276,85.391,-66.367,173.937,22.780,153.941
C00705=1078.282,85.641,-66.385,173.939,22.783,153.941
C00706=1078.287,85.890,-66.402,173.941,22.785,153.941
C00707=1078.293,86.140,-66.420,173.942,22.787,153.941
C00708=1078.299,86.389,-66.438,173.943,22.790,153.942
C00709=1078.305,86.638,-66.456,173.945,22.793,153.942
C00710=1078.311,86.888,-66.473,173.947,22.794,153.942
C00711=1078.316,87.137,-66.491,173.949,22.797,153.942
C00712=1078.322,87.387,-66.509,173.950,22.800,153.943
C00713=1078.328,87.636,-66.527,173.952,22.802,153.943
C00714=1078.333,87.885,-66.544,173.954,22.804,153.943
C00715=1078.339,88.135,-66.563,173.955,22.807,153.943
C00716=1078.345,88.383,-66.581,173.957,22.809,153.943
C00717=1078.351,88.633,-66.599,173.959,22.811,153.944
C00718=1078.356,88.882,-66.616,173.960,22.814,153.944
C00719=1078.362,89.132,-66.634,173.961,22.816,153.944
C00720=1078.368,89.381,-66.652,173.964,22.819,153.944
C00721=1078.374,89.630,-66.670,173.965,22.821,153.945
C00722=1078.379,89.879,-66.687,173.967,22.823,153.945
C00723=1078.386,90.129,-66.706,173.968,22.826,153.945
C00724=1078.391,90.378,-66.724,173.970,22.828,153.945
C00725=1078.398,90.627,-66.742,173.972,22.830,153.946
C00726=1078.403,90.876,-66.759,173.973,22.833,153.946
C00727=1078.408,91.126,-66.777,173.974,22.835,153.946
C00728=1078.414,91.375,-66.796,173.977,22.837,153.946
C00729=1078.420,91.624,-66.814,173.978,22.840,153.947
C00730=1078.425,91.874,-66.832,173.980,22.843,153.947
C00731=1078.431,92.123,-66.850,173.981,22.845,153.947
C00732=1078.437,92.372,-66.868,173.983,22.847,153.947
C00733=1078.443,92.621,-66.886,173.985,22.850,153.948
C00734=1078.448,92.871,-66.904,173.986,22.852,153.948
C00735=1078.454,93.120,-66.922,173.988,22.854,153.948
C00736=1078.459,93.369,-66.940,173.990,22.857,153.948
C00737=1078.465,93.619,-66.959,173.991,22.859,153.949
C00738=1078.470,93.868,-66.976,173.993,22.862,153.949
C00739=1078.477,94.117,-66.995,173.995,22.864,153.949
C00740=1078.482,94.366,-67.013,173.996,22.866,153.949
C00741=1078.488,94.616,-67.031,173.998,22.869,153.949
C00742=1078.494,94.896,-67.052,173.999,22.871,153.950
C00743=1078.500,95.177,-67.072,174.001,22.874,153.950
C00744=1078.507,95.457,-67.093,174.004,22.877,153.950
C00745=1078.513,95.738,-67.113,174.006,22.880,153.951
C00746=1078.520,95.987,-67.131,174.007,22.882,153.951
C00747=1078.524,96.237,-67.149,174.008,22.884,153.951
C00748=1078.531,96.486,-67.168,174.011,22.887,153.951
C00749=1078.536,96.735,-67.186,174.012,22.889,153.952
C00750=1078.542,96.984,-67.205,174.013,22.891,153.952
C00751=1078.547,97.233,-67.222,174.016,22.894,153.952
C00752=1078.554,97.483,-67.240,174.017,22.896,153.952
C00753=1078.559,97.732,-67.259,174.019,22.899,153.953
C00754=1078.565,97.982,-67.277,174.020,22.901,153.953
C00755=1078.571,98.231,-67.296,174.022,22.903,153.953
C00756=1078.576,98.480,-67.314,174.024,22.905,153.953
C00757=1078.582,98.729,-67.333,174.025,22.908,153.953
C00758=1078.587,98.979,-67.351,174.027,22.911,153.954
C00759=1078.594,99.228,-67.369,174.029,22.913,153.954
C00760=1078.599,99.477,-67.387,174.030,22.915,153.954
C00761=1078.605,99.726,-67.406,174.032,22.917,153.954
C00762=1078.611,99.976,-67.424,174.034,22.920,153.955
C00763=1078.617,100.224,-67.442,174.036,22.922,153.955
C00764=1078.622,100.474,-67.461,174.037,22.924,153.955
C00765=1078.628,100.723,-67.479,174.039,22.927,153.955
C00766=1078.633,100.973,-67.498,174.041,22.929,153.955
C00767=1078.640,101.222,-67.516,174.042,22.931,153.956
C00768=1078.645,101.471,-67.535,174.044,22.934,153.956
C00769=1078.651,101.720,-67.553,174.046,22.936,153.956
C00770=1078.656,101.969,-67.572,174.048,22.939,153.956
C00771=1078.662,102.219,-67.590,174.049,22.941,153.957
C00772=1078.668,102.468,-67.609,174.051,22.943,153.957
C00773=1078.674,102.717,-67.628,174.053,22.946,153.957
C00774=1078.679,102.967,-67.646,174.054,22.948,153.957
C00775=1078.684,103.216,-67.665,174.056,22.951,153.958
C00776=1078.690,103.465,-67.683,174.058,22.953,153.958
C00777=1078.695,103.714,-67.702,174.060,22.955,153.958
C00778=1078.702,103.963,-67.720,174.061,22.958,153.958
C00779=1078.707,104.213,-67.739,174.062,22.960,153.959
C00780=1078.712,104.462,-67.758,174.065,22.962,153.959
C00781=1078.719,104.711,-67.777,174.066,22.965,153.959
C00782=1078.724,104.960,-67.796,174.068,22.967,153.959
C00783=1078.730,105.209,-67.813,174.070,22.970,153.960
C00784=1078.736,105.459,-67.833,174.071,22.972,153.960
C00785=1078.741,105.708,-67.852,174.073,22.974,153.960
C00786=1078.747,105.957,-67.869,174.074,22.977,153.960
C00787=1078.752,106.207,-67.889,174.077,22.979,153.960
C00788=1078.758,106.456,-67.908,174.078,22.981,153.961
C00789=1078.764,106.705,-67.926,174.080,22.984,153.961
C00790=1078.769,106.955,-67.945,174.082,22.986,153.961
C00791=1078.775,107.203,-67.963,174.084,22.989,153.961
C00792=1078.781,107.453,-67.982,174.085,22.991,153.962
C00793=1078.787,107.702,-68.001,174.086,22.993,153.962
C00794=1078.793,107.951,-68.020,174.089,22.995,153.962
C00795=1078.798,108.201,-68.038,174.090,22.998,153.962
C00796=1078.803,108.450,-68.058,174.092,23.000,153.962
C00797=1078.810,108.699,-68.076,174.094,23.002,153.963
C00798=1078.815,108.948,-68.095,174.096,23.005,153.963
C00799=1078.821,109.197,-68.114,174.097,23.007,153.963
C00800=1078.827,109.446,-68.133,174.100,23.009,153.963
C00801=1078.832,109.696,-68.151,174.101,23.012,153.964
C00802=1078.838,109.945,-68.170,174.102,23.014,153.964
C00803=1078.844,110.194,-68.189,174.104,23.016,153.964
C00804=1078.850,110.444,-68.208,174.106,23.018,153.964
C00805=1078.855,110.692,-68.227,174.108,23.021,153.964
C00806=1078.862,110.973,-68.248,174.110,23.024,153.965
C00807=1078.868,111.254,-68.270,174.112,23.026,153.965
C00808=1078.875,111.535,-68.291,174.114,23.029,153.965
C00809=1078.881,111.815,-68.313,174.116,23.031,153.965
C00810=1078.886,112.065,-68.331,174.117,23.034,153.966
C00811=1078.893,112.314,-68.350,174.120,23.036,153.966
C00812=1078.898,112.563,-68.369,174.121,23.038,153.966
C00813=1078.904,112.812,-68.388,174.123,23.041,153.966
C00814=1078.909,113.062,-68.407,174.124,23.043,153.967
C00815=1078.915,113.311,-68.427,174.127,23.045,153.967
C00816=1078.921,113.559,-68.445,174.128,23.048,153.967
C00817=1078.926,113.809,-68.464,174.130,23.050,153.967
C00818=1078.932,114.058,-68.483,174.132,23.052,153.967
C00819=1078.938,114.308,-68.503,174.133,23.054,153.968
C00820=1078.943,114.557,-68.522,174.135,23.057,153.968
C00821=1078.949,114.805,-68.541,174.137,23.059,153.968
C00822=1078.955,115.055,-68.561,174.139,23.062,153.968
C00823=1078.960,115.304,-68.580,174.140,23.064,153.969
C00824=1078.965,115.553,-68.599,174.142,23.066,153.969
C00825=1078.971,115.802,-68.618,174.144,23.069,153.969
C00826=1078.977,116.052,-68.637,174.146,23.071,153.969
C00827=1078.982,116.301,-68.656,174.147,23.073,153.969
C00828=1078.987,116.550,-68.675,174.150,23.076,153.970
C00829=1078.993,116.799,-68.695,174.151,23.078,153.970
C00830=1078.999,117.049,-68.714,174.153,23.081,153.970
C00831=1079.005,117.298,-68.733,174.155,23.083,153.970
C00832=1079.010,117.546,-68.753,174.157,23.086,153.971
C00833=1079.016,117.796,-68.772,174.158,23.087,153.971
C00834=1079.021,118.045,-68.791,174.160,23.090,153.971
C00835=1079.027,118.295,-68.810,174.162,23.092,153.971
C00836=1079.033,118.544,-68.830,174.164,23.095,153.971
C00837=1079.038,118.792,-68.849,174.165,23.097,153.972
C00838=1079.044,119.042,-68.868,174.168,23.099,153.972
C00839=1079.049,119.291,-68.888,174.169,23.101,153.972
C00840=1079.055,119.541,-68.907,174.170,23.104,153.972
C00841=1079.061,119.790,-68.926,174.173,23.106,153.972
C00842=1079.067,120.039,-68.946,174.174,23.108,153.973
C00843=1079.071,120.288,-68.966,174.176,23.111,153.973
C00844=1079.077,120.537,-68.985,174.178,23.113,153.973
C00845=1079.083,120.787,-69.004,174.180,23.115,153.973
C00846=1079.089,121.035,-69.024,174.181,23.118,153.974
C00847=1079.094,121.285,-69.043,174.183,23.120,153.974
C00848=1079.100,121.534,-69.063,174.185,23.122,153.974
C00849=1079.105,121.782,-69.082,174.187,23.125,153.974
C00850=1079.111,122.032,-69.101,174.188,23.127,153.974
C00851=1079.117,122.281,-69.121,174.191,23.129,153.975
C00852=1079.123,122.530,-69.141,174.192,23.132,153.975
C00853=1079.128,122.780,-69.160,174.194,23.134,153.975
C00854=1079.134,123.029,-69.179,174.196,23.136,153.975
C00855=1079.139,123.278,-69.200,174.198,23.139,153.975
C00856=1079.145,123.528,-69.219,174.200,23.141,153.976
C00857=1079.151,123.777,-69.238,174.202,23.143,153.976
C00858=1079.156,124.025,-69.258,174.204,23.145,153.976
C00859=1079.162,124.275,-69.277,174.205,23.148,153.976
C00860=1079.167,124.524,-69.296,174.208,23.150,153.976
C00861=1079.173,124.773,-69.316,174.209,23.153,153.977
C00862=1079.179,125.022,-69.335,174.211,23.155,153.977
C00863=1079.184,125.271,-69.356,174.213,23.157,153.977
C00864=1079.190,125.521,-69.375,174.215,23.159,153.977
C00865=1079.196,125.770,-69.395,174.216,23.161,153.977
C00866=1079.202,126.019,-69.414,174.219,23.164,153.978
C00867=1079.208,126.268,-69.434,174.220,23.166,153.978
C00868=1079.213,126.517,-69.454,174.222,23.168,153.978
C00869=1079.219,126.766,-69.474,174.223,23.171,153.978
C00870=1079.226,127.047,-69.495,174.226,23.173,153.978
C00871=1079.231,127.328,-69.518,174.228,23.176,153.979
C00872=1079.238,127.608,-69.540,174.230,23.178,153.979
C00873=1079.245,127.889,-69.563,174.232,23.181,153.979
C00874=1079.250,128.138,-69.582,174.234,23.183,153.979
C00875=1079.256,128.387,-69.602,174.236,23.185,153.980
C00876=1079.262,128.637,-69.621,174.238,23.187,153.980
C00877=1079.268,128.885,-69.641,174.240,23.190,153.980
C00878=1079.274,129.135,-69.660,174.241,23.192,153.980
C00879=1079.279,129.384,-69.681,174.244,23.194,153.980
C00880=1079.285,129.633,-69.701,174.245,23.196,153.981
C00881=1079.291,129.882,-69.720,174.247,23.199,153.981
C00882=1079.297,130.131,-69.740,174.249,23.201,153.981
C00883=1079.302,130.380,-69.759,174.251,23.203,153.981
C00884=1079.308,130.630,-69.780,174.253,23.206,153.981
C00885=1079.314,130.878,-69.800,174.255,23.207,153.981
C00886=1079.319,131.128,-69.819,174.257,23.210,153.982
C00887=1079.325,131.377,-69.839,174.258,23.212,153.982
C00888=1079.330,131.626,-69.860,174.261,23.214,153.982
C00889=1079.336,131.875,-69.879,174.262,23.216,153.982
C00890=1079.342,132.124,-69.899,174.264,23.218,153.982
C00891=1079.348,132.373,-69.919,174.266,23.221,153.983
C00892=1079.353,132.623,-69.939,174.268,23.223,153.983
C00893=1079.360,132.872,-69.959,174.270,23.226,153.983
C00894=1079.365,133.121,-69.980,174.272,23.228,153.983
C00895=1079.371,133.370,-70.000,174.274,23.230,153.983
C00896=1079.376,133.620,-70.019,174.275,23.232,153.984
C00897=1079.382,133.869,-70.039,174.278,23.235,153.984
C00898=1079.388,134.117,-70.059,174.279,23.236,153.984
C00899=1079.393,134.367,-70.080,174.281,23.239,153.984
C00900=1079.399,134.616,-70.099,174.284,23.242,153.984
C00901=1079.404,134.865,-70.120,174.285,23.243,153.985
C00902=1079.410,135.114,-70.140,174.287,23.246,153.985
C00903=1079.415,135.363,-70.160,174.289,23.248,153.985
C00904=1079.421,135.612,-70.180,174.291,23.250,153.985
C00905=1079.426,135.862,-70.200,174.292,23.253,153.985
C00906=1079.432,136.110,-70.220,174.295,23.255,153.986
C00907=1079.438,136.360,-70.240,174.297,23.257,153.986
C00908=1079.444,136.608,-70.260,174.298,23.260,153.986
C00909=1079.449,136.858,-70.281,174.301,23.262,153.986
C00910=1079.455,137.107,-70.301,174.302,23.264,153.986
C00911=1079.461,137.356,-70.322,174.304,23.266,153.987
C00912=1079.466,137.606,-70.341,174.306,23.268,153.987
C00913=1079.472,137.855,-70.362,174.308,23.271,153.987
C00914=1079.478,138.103,-70.382,174.310,23.273,153.987
C00915=1079.483,138.353,-70.402,174.312,23.275,153.987
C00916=1079.489,138.601,-70.422,174.314,23.277,153.987
C00917=1079.494,138.851,-70.443,174.315,23.280,153.988
C00918=1079.501,139.100,-70.463,174.318,23.282,153.988
C00919=1079.506,139.349,-70.484,174.320,23.284,153.988
C00920=1079.512,139.598,-70.504,174.321,23.286,153.988
C00921=1079.517,139.847,-70.524,174.324,23.289,153.988
C00922=1079.523,140.096,-70.544,174.325,23.291,153.989
C00923=1079.528,140.345,-70.565,174.327,23.293,153.989
C00924=1079.534,140.594,-70.585,174.330,23.296,153.989
C00925=1079.540,140.844,-70.605,174.331,23.298,153.989
C00926=1079.546,141.093,-70.626,174.333,23.300,153.989
C00927=1079.551,141.342,-70.647,174.335,23.302,153.990
C00928=1079.557,141.591,-70.667,174.337,23.305,153.990
C00929=1079.562,141.840,-70.687,174.339,23.307,153.990
C00930=1079.567,142.089,-70.708,174.341,23.309,153.990
C00931=1079.573,142.338,-70.728,174.343,23.311,153.990
C00932=1079.579,142.588,-70.749,174.345,23.313,153.990
C00933=1079.584,142.837,-70.769,174.347,23.315,153.991
C00934=1079.591,143.117,-70.793,174.349,23.318,153.991
C00935=1079.597,143.398,-70.815,174.351,23.321,153.991
C00936=1079.604,143.678,-70.839,174.354,23.323,153.991
C00937=1079.610,143.958,-70.861,174.356,23.326,153.992
C00938=1079.616,144.208,-70.882,174.357,23.328,153.992
C00939=1079.621,144.456,-70.903,174.360,23.330,153.992
C00940=1079.626,144.706,-70.924,174.362,23.332,153.992
C00941=1079.632,144.954,-70.944,174.363,23.335,153.992
C00942=1079.638,145.204,-70.965,174.366,23.337,153.992
C00943=1079.644,145.453,-70.985,174.368,23.339,153.993
C00944=1079.649,145.702,-71.006,174.369,23.341,153.993
C00945=1079.655,145.951,-71.026,174.372,23.344,153.993
C00946=1079.660,146.200,-71.047,174.373,23.346,153.993
C00947=1079.666,146.450,-71.068,174.375,23.348,153.993
C00948=1079.671,146.699,-71.088,174.378,23.350,153.993
C00949=1079.678,146.947,-71.109,174.379,23.353,153.994
C00950=1079.684,147.197,-71.130,174.381,23.355,153.994
C00951=1079.689,147.446,-71.151,174.384,23.357,153.994
C00952=1079.694,147.695,-71.171,174.385,23.359,153.994
C00953=1079.700,147.943,-71.192,174.388,23.361,153.994
C00954=1079.706,148.193,-71.213,174.390,23.364,153.995
C00955=1079.712,148.442,-71.233,174.391,23.366,153.995
C00956=1079.717,148.691,-71.255,174.394,23.368,153.995
C00957=1079.722,148.940,-71.275,174.396,23.370,153.995
C00958=1079.728,149.190,-71.296,174.397,23.373,153.995
C00959=1079.734,149.438,-71.317,174.400,23.375,153.995
C00960=1079.739,149.687,-71.338,174.401,23.377,153.996
C00961=1079.746,149.937,-71.358,174.403,23.379,153.996
C00962=1079.751,150.185,-71.379,174.406,23.382,153.996
C00963=1079.756,150.434,-71.400,174.407,23.384,153.996
C00964=1079.762,150.683,-71.421,174.409,23.386,153.996
C00965=1079.768,150.933,-71.442,174.412,23.388,153.996
C00966=1079.773,151.182,-71.463,174.413,23.390,153.997
C00967=1079.779,151.430,-71.484,174.415,23.393,153.997
C00968=1079.785,151.680,-71.505,174.418,23.395,153.997
C00969=1079.790,151.929,-71.526,174.419,23.397,153.997
C00970=1079.795,152.178,-71.547,174.422,23.399,153.997
C00971=1079.802,152.427,-71.568,174.424,23.402,153.998
C00972=1079.807,152.676,-71.589,174.425,23.404,153.998
C00973=1079.812,152.925,-71.610,174.428,23.406,153.998
C00974=1079.818,153.174,-71.631,174.430,23.408,153.998
C00975=1079.824,153.423,-71.652,174.431,23.410,153.998
C00976=1079.829,153.672,-71.673,174.434,23.413,153.999
C00977=1079.835,153.921,-71.695,174.436,23.415,153.999
C00978=1079.840,154.170,-71.715,174.438,23.417,153.999
C00979=1079.846,154.419,-71.736,174.440,23.419,153.999
C00980=1079.852,154.669,-71.757,174.442,23.422,153.999
C00981=1079.857,154.917,-71.779,174.444,23.424,153.999
C00982=1079.863,155.166,-71.799,174.446,23.426,154.000
C00983=1079.869,155.415,-71.821,174.448,23.428,154.000
C00984=1079.874,155.664,-71.842,174.451,23.430,154.000
C00985=1079.880,155.914,-71.863,174.452,23.432,154.000
C00986=1079.886,156.162,-71.884,174.454,23.435,154.000
C00987=1079.891,156.411,-71.905,174.457,23.437,154.000
C00988=1079.896,156.661,-71.927,174.458,23.439,154.001
C00989=1079.902,156.909,-71.948,174.460,23.441,154.001
C00990=1079.907,157.159,-71.969,174.463,23.444,154.001
C00991=1079.913,157.408,-71.991,174.465,23.446,154.001
C00992=1079.919,157.656,-72.012,174.466,23.448,154.001
C00993=1079.925,157.906,-72.033,174.469,23.450,154.001
C00994=1079.930,158.155,-72.054,174.471,23.453,154.002
C00995=1079.936,158.403,-72.075,174.473,23.454,154.002
C00996=1079.941,158.653,-72.097,174.475,23.457,154.002
C00997=1079.947,158.902,-72.118,174.477,23.459,154.002
C00998=1079.953,159.182,-72.142,174.480,23.462,154.002
C00999=1079.960,159.462,-72.166,174.482,23.464,154.003
C01000=1079.966,159.743,-72.190,174.484,23.467,154.003
C01001=1079.973,160.023,-72.214,174.487,23.469,154.003
C01002=1079.978,160.272,-72.235,174.489,23.472,154.003
C01003=1079.984,160.521,-72.258,174.490,23.474,154.003
C01004=1079.989,160.770,-72.279,174.493,23.476,154.003
C01005=1079.995,161.020,-72.300,174.495,23.478,154.004
C01006=1080.001,161.268,-72.321,174.497,23.480,154.004
C01007=1080.006,161.517,-72.342,174.499,23.482,154.004
C01008=1080.012,161.766,-72.365,174.501,23.485,154.004
C01009=1080.017,162.015,-72.386,174.503,23.487,154.004
C01010=1080.023,162.264,-72.408,174.506,23.489,154.004
C01011=1080.028,162.513,-72.429,174.507,23.491,154.005
C01012=1080.033,162.762,-72.450,174.509,23.494,154.005
C01013=1080.039,163.011,-72.472,174.512,23.496,154.005
C01014=1080.044,163.260,-72.494,174.514,23.498,154.005
C01015=1080.050,163.509,-72.516,174.515,23.501,154.005
C01016=1080.055,163.758,-72.537,174.518,23.503,154.006
C01017=1080.061,164.007,-72.559,174.520,23.505,154.006
C01018=1080.066,164.256,-72.580,174.523,23.507,154.006
C01019=1080.071,164.505,-72.602,174.524,23.510,154.006
C01020=1080.077,164.754,-72.624,174.526,23.512,154.006
C01021=1080.082,165.003,-72.646,174.529,23.514,154.006
C01022=1080.088,165.252,-72.667,174.531,23.516,154.007
C01023=1080.093,165.501,-72.689,174.532,23.519,154.007
C01024=1080.099,165.750,-72.711,174.535,23.521,154.007
C01025=1080.104,165.999,-72.733,174.537,23.523,154.007
C01026=1080.110,166.248,-72.754,174.539,23.526,154.007
C01027=1080.115,166.497,-72.776,174.541,23.527,154.007
C01028=1080.121,166.746,-72.798,174.543,23.530,154.008
C01029=1080.126,166.995,-72.820,174.545,23.532,154.008
C01030=1080.132,167.244,-72.842,174.548,23.535,154.008
C01031=1080.137,167.493,-72.863,174.549,23.536,154.008
C01032=1080.143,167.742,-72.885,174.551,23.539,154.008
C01033=1080.148,167.991,-72.907,174.554,23.541,154.009
C01034=1080.154,168.240,-72.929,174.556,23.544,154.009
C01035=1080.159,168.489,-72.950,174.559,23.546,154.009
C01036=1080.165,168.738,-72.973,174.560,23.548,154.009
C01037=1080.170,168.986,-72.994,174.562,23.550,154.009
C01038=1080.176,169.236,-73.017,174.565,23.553,154.009
C01039=1080.182,169.485,-73.038,174.567,23.555,154.010
C01040=1080.187,169.734,-73.060,174.568,23.557,154.010
C01041=1080.192,169.983,-73.082,174.571,23.559,154.010
C01042=1080.198,170.232,-73.104,174.573,23.561,154.010
C01043=1080.204,170.481,-73.127,174.575,23.563,154.010
C01044=1080.209,170.729,-73.148,174.578,23.566,154.010
C01045=1080.215,170.979,-73.170,174.579,23.568,154.011
C01046=1080.221,171.228,-73.192,174.582,23.570,154.011
C01047=1080.226,171.476,-73.214,174.584,23.572,154.011
C01048=1080.231,171.726,-73.237,174.586,23.575,154.011
C01049=1080.237,171.974,-73.258,174.589,23.577,154.011
C01050=1080.242,172.224,-73.280,174.590,23.579,154.011
C01051=1080.249,172.472,-73.302,174.592,23.582,154.012
C01052=1080.254,172.721,-73.324,174.595,23.584,154.012
C01053=1080.259,172.971,-73.346,174.597,23.586,154.012
C01054=1080.265,173.219,-73.369,174.599,23.588,154.012
C01055=1080.270,173.468,-73.391,174.601,23.590,154.012
C01056=1080.276,173.717,-73.412,174.603,23.592,154.012
C01057=1080.282,173.967,-73.435,174.606,23.594,154.012
C01058=1080.287,174.215,-73.457,174.608,23.597,154.013
C01059=1080.293,174.464,-73.479,174.610,23.599,154.013
C01060=1080.299,174.713,-73.502,174.613,23.602,154.013
C01061=1080.304,174.962,-73.524,174.614,23.604,154.013
C01062=1080.310,175.241,-73.548,174.617,23.606,154.013
C01063=1080.317,175.522,-73.573,174.620,23.608,154.013
C01064=1080.323,175.802,-73.598,174.622,23.611,154.014
C01065=1080.329,176.081,-73.624,174.624,23.613,154.014
C01066=1080.336,176.331,-73.645,174.627,23.616,154.014
C01067=1080.341,176.579,-73.668,174.629,23.618,154.014
C01068=1080.346,176.828,-73.690,174.631,23.620,154.014
C01069=1080.352,177.077,-73.712,174.633,23.622,154.014
C01070=1080.358,177.326,-73.735,174.635,23.624,154.015
C01071=1080.363,177.575,-73.757,174.638,23.626,154.015
C01072=1080.369,177.824,-73.779,174.640,23.629,154.015
C01073=1080.375,178.073,-73.801,174.642,23.631,154.015
C01074=1080.380,178.322,-73.824,174.645,23.633,154.015
C01075=1080.386,178.570,-73.847,174.647,23.635,154.015
C01076=1080.392,178.820,-73.868,174.649,23.637,154.015
C01077=1080.398,179.068,-73.891,174.651,23.639,154.016
C01078=1080.403,179.318,-73.913,174.653,23.642,154.016
C01079=1080.409,179.567,-73.936,174.656,23.644,154.016
C01080=1080.414,179.815,-73.958,174.658,23.646,154.016
C01081=1080.420,180.064,-73.981,174.660,23.649,154.016
C01082=1080.426,180.313,-74.004,174.663,23.651,154.016
C01083=1080.432,180.562,-74.025,174.664,23.653,154.017
C01084=1080.438,180.811,-74.048,174.667,23.655,154.017
C01085=1080.443,181.061,-74.070,174.669,23.657,154.017
C01086=1080.448,181.309,-74.093,174.671,23.659,154.017
C01087=1080.455,181.558,-74.115,174.674,23.662,154.017
C01088=1080.460,181.807,-74.138,174.676,23.664,154.017
C01089=1080.466,182.056,-74.160,174.679,23.665,154.017
C01090=1080.472,182.305,-74.183,174.681,23.668,154.017
C01091=1080.478,182.554,-74.205,174.683,23.670,154.018
C01092=1080.483,182.803,-74.228,174.685,23.672,154.018
C01093=1080.489,183.051,-74.251,174.687,23.674,154.018
C01094=1080.494,183.300,-74.274,174.690,23.676,154.018
C01095=1080.500,183.549,-74.295,174.692,23.678,154.018
C01096=1080.506,183.798,-74.318,174.694,23.681,154.018
C01097=1080.512,184.047,-74.341,174.697,23.683,154.019
C01098=1080.518,184.296,-74.364,174.699,23.685,154.019
C01099=1080.524,184.545,-74.386,174.702,23.687,154.019
C01100=1080.530,184.794,-74.409,174.704,23.690,154.019
C01101=1080.535,185.043,-74.432,174.705,23.691,154.019
C01102=1080.540,185.291,-74.454,174.708,23.694,154.019
C01103=1080.546,185.540,-74.477,174.710,23.696,154.019
C01104=1080.551,185.789,-74.501,174.712,23.699,154.020
C01105=1080.557,186.039,-74.523,174.715,23.701,154.020
C01106=1080.562,186.288,-74.546,174.717,23.703,154.020
C01107=1080.567,186.536,-74.568,174.720,23.705,154.020
C01108=1080.573,186.785,-74.591,174.722,23.707,154.020
C01109=1080.579,187.034,-74.614,174.724,23.710,154.021
C01110=1080.584,187.283,-74.638,174.726,23.712,154.021
C01111=1080.590,187.532,-74.661,174.729,23.715,154.021
C01112=1080.595,187.781,-74.684,174.730,23.716,154.021
C01113=1080.600,188.029,-74.706,174.733,23.719,154.021
C01114=1080.606,188.278,-74.729,174.735,23.721,154.021
C01115=1080.612,188.527,-74.752,174.737,23.724,154.022
C01116=1080.617,188.776,-74.776,174.740,23.726,154.022
C01117=1080.622,189.025,-74.798,174.742,23.728,154.022
C01118=1080.628,189.274,-74.821,174.744,23.730,154.022
C01119=1080.634,189.523,-74.844,174.747,23.732,154.022
C01120=1080.640,189.771,-74.867,174.749,23.735,154.022
C01121=1080.644,190.020,-74.891,174.752,23.737,154.022
C01122=1080.650,190.269,-74.914,174.754,23.740,154.023
C01123=1080.656,190.518,-74.937,174.756,23.742,154.023
C01124=1080.661,190.767,-74.960,174.759,23.744,154.023
C01125=1080.666,191.016,-74.983,174.761,23.746,154.023
C01126=1080.673,191.295,-75.009,174.763,23.748,154.023
C01127=1080.679,191.575,-75.035,174.766,23.751,154.023
C01128=1080.685,191.855,-75.061,174.769,23.754,154.024
C01129=1080.692,192.134,-75.086,174.771,23.757,154.024
C01130=1080.697,192.383,-75.109,174.773,23.759,154.024
C01131=1080.702,192.632,-75.133,174.776,23.761,154.024
C01132=1080.708,192.881,-75.157,174.778,23.763,154.024
C01133=1080.714,193.129,-75.180,174.781,23.765,154.024
C01134=1080.720,193.378,-75.203,174.783,23.768,154.025
C01135=1080.725,193.628,-75.226,174.785,23.770,154.025
C01136=1080.731,193.877,-75.249,174.788,23.772,154.025
C01137=1080.736,194.125,-75.272,174.790,23.774,154.025
C01138=1080.742,194.374,-75.296,174.793,23.776,154.025
C01139=1080.747,194.623,-75.319,174.795,23.779,154.025
C01140=1080.753,194.872,-75.342,174.797,23.781,154.026
C01141=1080.759,195.121,-75.365,174.800,23.784,154.026
C01142=1080.764,195.369,-75.389,174.802,23.786,154.026
C01143=1080.770,195.618,-75.412,174.804,23.788,154.026
C01144=1080.775,195.867,-75.435,174.807,23.790,154.026
C01145=1080.781,196.116,-75.459,174.809,23.792,154.026
C01146=1080.787,196.365,-75.482,174.811,23.795,154.026
C01147=1080.792,196.613,-75.505,174.814,23.797,154.027
C01148=1080.797,196.863,-75.529,174.816,23.799,154.027
C01149=1080.803,197.111,-75.553,174.819,23.801,154.027
C01150=1080.809,197.360,-75.575,174.821,23.803,154.027
C01151=1080.814,197.608,-75.600,174.823,23.806,154.027
C01152=1080.820,197.857,-75.623,174.826,23.808,154.027
C01153=1080.826,198.107,-75.646,174.828,23.810,154.027
C01154=1080.832,198.355,-75.670,174.831,23.812,154.028
C01155=1080.837,198.604,-75.693,174.833,23.815,154.028
C01156=1080.843,198.853,-75.716,174.835,23.817,154.028
C01157=1080.848,199.102,-75.740,174.838,23.819,154.028
C01158=1080.854,199.351,-75.763,174.840,23.822,154.028
C01159=1080.860,199.599,-75.787,174.842,23.824,154.028
C01160=1080.865,199.848,-75.811,174.845,23.826,154.029
C01161=1080.872,200.097,-75.835,174.847,23.828,154.029
C01162=1080.878,200.346,-75.858,174.850,23.830,154.029
C01163=1080.883,200.595,-75.882,174.852,23.833,154.029
C01164=1080.889,200.844,-75.905,174.854,23.835,154.029
C01165=1080.894,201.092,-75.929,174.857,23.837,154.029
C01166=1080.900,201.341,-75.952,174.859,23.839,154.029
C01167=1080.906,201.590,-75.976,174.861,23.842,154.030
C01168=1080.911,201.839,-75.999,174.864,23.844,154.030
C01169=1080.917,202.088,-76.023,174.866,23.846,154.030
C01170=1080.922,202.337,-76.047,174.869,23.848,154.030
C01171=1080.928,202.585,-76.070,174.871,23.850,154.030
C01172=1080.934,202.834,-76.095,174.873,23.853,154.030
C01173=1080.940,203.083,-76.118,174.876,23.855,154.030
C01174=1080.945,203.332,-76.142,174.878,23.857,154.031
C01175=1080.951,203.580,-76.166,174.880,23.860,154.031
C01176=1080.956,203.829,-76.189,174.883,23.862,154.031
C01177=1080.962,204.078,-76.214,174.885,23.864,154.031
C01178=1080.967,204.327,-76.237,174.889,23.867,154.031
C01179=1080.973,204.576,-76.261,174.891,23.869,154.031
C01180=1080.979,204.825,-76.285,174.893,23.871,154.032
C01181=1080.985,205.073,-76.309,174.896,23.873,154.032
C01182=1080.990,205.322,-76.333,174.898,23.876,154.032
C01183=1080.995,205.571,-76.357,174.900,23.878,154.032
C01184=1081.001,205.819,-76.381,174.903,23.880,154.032
C01185=1081.006,206.069,-76.404,174.905,23.883,154.032
C01186=1081.012,206.318,-76.429,174.907,23.885,154.033
C01187=1081.018,206.566,-76.452,174.910,23.887,154.033
C01188=1081.023,206.814,-76.477,174.912,23.889,154.033
C01189=1081.029,207.064,-76.501,174.915,23.891,154.033
C01190=1081.052,208.096,-76.600,175.012,23.943,154.031
C01191=1081.061,208.494,-76.640,175.016,23.948,154.032
C01192=1081.071,208.891,-76.679,175.019,23.954,154.032
C01193=1081.080,209.288,-76.718,175.023,23.959,154.033
C01194=1081.089,209.686,-76.757,175.027,23.964,154.034
C01195=1081.094,209.934,-76.781,175.029,23.968,154.034
C01196=1081.100,210.183,-76.807,175.032,23.971,154.034
C01197=1081.106,210.432,-76.831,175.034,23.974,154.035
C01198=1081.111,210.681,-76.856,175.036,23.977,154.035
C01199=1081.117,210.929,-76.881,175.039,23.980,154.035
C01200=1081.123,211.178,-76.905,175.041,23.984,154.036
C01201=1081.128,211.427,-76.929,175.043,23.987,154.036
C01202=1081.134,211.676,-76.955,175.045,23.990,154.037
C01203=1081.140,211.924,-76.979,175.048,23.994,154.037
C01204=1081.145,212.174,-77.004,175.050,23.996,154.037
C01205=1081.151,212.422,-77.029,175.052,24.000,154.038
C01206=1081.156,212.671,-77.054,175.055,24.003,154.038
C01207=1081.162,212.919,-77.079,175.057,24.007,154.038
C01208=1081.168,213.168,-77.103,175.060,24.010,154.039
C01209=1081.174,213.416,-77.128,175.062,24.013,154.039
C01210=1081.179,213.666,-77.153,175.065,24.017,154.040
C01211=1081.185,213.914,-77.177,175.067,24.020,154.040
C01212=1081.190,214.163,-77.203,175.069,24.023,154.040
C01213=1081.195,214.412,-77.227,175.071,24.026,154.041
C01214=1081.202,214.660,-77.253,175.074,24.029,154.041
C01215=1081.208,214.909,-77.278,175.076,24.033,154.042
C01216=1081.213,215.158,-77.302,175.078,24.036,154.042
C01217=1081.219,215.407,-77.328,175.081,24.039,154.042
C01218=1081.224,215.655,-77.353,175.083,24.043,154.043
C01219=1081.230,215.904,-77.378,175.085,24.046,154.043
C01220=1081.235,216.152,-77.402,175.087,24.049,154.044
C01221=1081.242,216.401,-77.428,175.091,24.052,154.044
C01222=1081.247,216.649,-77.453,175.093,24.055,154.044
C01223=1081.252,216.899,-77.478,175.095,24.059,154.045
C01224=1081.259,217.147,-77.503,175.098,24.062,154.045
C01225=1081.264,217.396,-77.527,175.100,24.065,154.045
C01226=1081.269,217.645,-77.553,175.102,24.069,154.046
C01227=1081.276,217.894,-77.579,175.104,24.072,154.046
C01228=1081.281,218.142,-77.603,175.107,24.075,154.046
C01229=1081.287,218.391,-77.628,175.109,24.078,154.047
C01230=1081.292,218.639,-77.654,175.111,24.081,154.047
C01231=1081.298,218.888,-77.679,175.114,24.085,154.048
C01232=1081.304,219.137,-77.704,175.116,24.088,154.048
C01233=1081.309,219.385,-77.729,175.119,24.091,154.048
C01234=1081.315,219.634,-77.755,175.121,24.094,154.049
C01235=1081.321,219.883,-77.780,175.124,24.098,154.049
C01236=1081.327,220.131,-77.804,175.126,24.101,154.050
C01237=1081.332,220.380,-77.830,175.128,24.104,154.050
C01238=1081.338,220.629,-77.855,175.131,24.108,154.050
C01239=1081.344,220.877,-77.880,175.133,24.110,154.051
C01240=1081.349,221.126,-77.906,175.135,24.114,154.051
C01241=1081.356,221.375,-77.932,175.138,24.117,154.051
C01242=1081.362,221.624,-77.956,175.140,24.121,154.052
C01243=1081.370,222.025,-77.998,175.144,24.126,154.052
C01244=1081.380,222.426,-78.039,175.148,24.131,154.053
C01245=1081.388,222.828,-78.080,175.152,24.136,154.054
C01246=1081.398,223.229,-78.121,175.155,24.141,154.054
C01247=1081.403,223.478,-78.146,175.158,24.145,154.055
C01248=1081.409,223.727,-78.172,175.161,24.148,154.055
C01249=1081.414,223.976,-78.198,175.163,24.151,154.056
C01250=1081.420,224.224,-78.222,175.166,24.155,154.056
C01251=1081.425,224.473,-78.248,175.168,24.158,154.056
C01252=1081.432,224.721,-78.274,175.170,24.161,154.057
C01253=1081.437,224.970,-78.300,175.173,24.165,154.057
C01254=1081.442,225.219,-78.325,175.175,24.168,154.057
C01255=1081.448,225.467,-78.351,175.177,24.171,154.058
C01256=1081.454,225.716,-78.377,175.180,24.175,154.058
C01257=1081.460,225.964,-78.403,175.182,24.177,154.058
C01258=1081.465,226.213,-78.428,175.185,24.181,154.059
C01259=1081.471,226.461,-78.453,175.188,24.184,154.059
C01260=1081.477,226.710,-78.479,175.190,24.187,154.060
C01261=1081.483,226.959,-78.505,175.193,24.191,154.060
C01262=1081.488,227.208,-78.531,175.195,24.194,154.060
C01263=1081.494,227.457,-78.557,175.197,24.197,154.061
C01264=1081.500,227.704,-78.582,175.200,24.200,154.061
C01265=1081.505,227.953,-78.608,175.202,24.204,154.062
C01266=1081.511,228.202,-78.634,175.204,24.207,154.062
C01267=1081.517,228.451,-78.660,175.207,24.210,154.062
C01268=1081.522,228.700,-78.685,175.209,24.214,154.063
C01269=1081.529,228.948,-78.711,175.211,24.217,154.063
C01270=1081.534,229.196,-78.737,175.215,24.220,154.063
C01271=1081.539,229.445,-78.763,175.217,24.223,154.064
C01272=1081.545,229.694,-78.788,175.220,24.227,154.064
C01273=1081.551,229.942,-78.815,175.222,24.230,154.065
C01274=1081.557,230.191,-78.840,175.224,24.233,154.065
C01275=1081.563,230.440,-78.866,175.227,24.236,154.065
C01276=1081.569,230.688,-78.893,175.229,24.239,154.066
C01277=1081.573,230.936,-78.918,175.231,24.243,154.066
C01278=1081.580,231.185,-78.944,175.234,24.246,154.066
C01279=1081.585,231.433,-78.970,175.236,24.249,154.067
C01280=1081.591,231.682,-78.996,175.239,24.253,154.067
C01281=1081.596,231.931,-79.022,175.242,24.256,154.068
C01282=1081.602,232.180,-79.049,175.244,24.259,154.068
C01283=1081.608,232.429,-79.075,175.247,24.263,154.068
C01284=1081.614,232.677,-79.101,175.249,24.266,154.069
C01285=1081.620,232.926,-79.127,175.251,24.269,154.069
C01286=1081.624,233.174,-79.152,175.254,24.272,154.069
C01287=1081.630,233.422,-79.179,175.256,24.276,154.070
C01288=1081.636,233.671,-79.205,175.259,24.279,154.070
C01289=1081.641,233.920,-79.232,175.261,24.282,154.071
C01290=1081.648,234.168,-79.257,175.263,24.286,154.071
C01291=1081.653,234.417,-79.284,175.266,24.289,154.071
C01292=1081.659,234.666,-79.310,175.268,24.292,154.072
C01293=1081.665,234.914,-79.336,175.272,24.295,154.072
C01294=1081.670,235.163,-79.362,175.274,24.299,154.073
C01295=1081.679,235.556,-79.404,175.277,24.304,154.073
C01296=1081.687,235.949,-79.446,175.282,24.309,154.074
C01297=1081.697,236.342,-79.487,175.285,24.314,154.074
C01298=1081.706,236.735,-79.529,175.290,24.320,154.075
C01299=1081.712,236.983,-79.555,175.292,24.323,154.075
C01300=1081.717,237.231,-79.582,175.294,24.326,154.076
C01301=1081.723,237.480,-79.608,175.297,24.330,154.076
C01302=1081.729,237.729,-79.635,175.299,24.333,154.077
C01303=1081.734,237.977,-79.661,175.302,24.336,154.077
C01304=1081.740,238.226,-79.687,175.305,24.339,154.077
C01305=1081.746,238.474,-79.714,175.308,24.343,154.078
C01306=1081.751,238.723,-79.741,175.310,24.346,154.078
C01307=1081.757,238.971,-79.767,175.312,24.349,154.079
C01308=1081.763,239.220,-79.793,175.315,24.353,154.079
C01309=1081.768,239.468,-79.820,175.317,24.356,154.079
C01310=1081.774,239.717,-79.846,175.320,24.359,154.080
C01311=1081.780,239.965,-79.873,175.322,24.362,154.080
C01312=1081.786,240.215,-79.899,175.325,24.366,154.080
C01313=1081.792,240.463,-79.926,175.327,24.369,154.081
C01314=1081.798,240.712,-79.953,175.330,24.372,154.081
C01315=1081.803,240.960,-79.979,175.333,24.376,154.082
C01316=1081.809,241.208,-80.006,175.335,24.379,154.082
C01317=1081.814,241.457,-80.033,175.338,24.382,154.082
C01318=1081.820,241.705,-80.060,175.340,24.386,154.083
C01319=1081.826,241.954,-80.086,175.343,24.389,154.083
C01320=1081.831,242.203,-80.112,175.345,24.392,154.083
C01321=1081.837,242.451,-80.139,175.348,24.395,154.084
C01322=1081.843,242.700,-80.166,175.350,24.399,154.084
C01323=1081.849,242.948,-80.193,175.353,24.402,154.085
C01324=1081.855,243.197,-80.219,175.355,24.405,154.085
C01325=1081.860,243.446,-80.247,175.358,24.408,154.085
C01326=1081.866,243.694,-80.273,175.361,24.412,154.086
C01327=1081.871,243.942,-80.300,175.363,24.415,154.086
C01328=1081.876,244.191,-80.327,175.366,24.419,154.087
C01329=1081.882,244.439,-80.354,175.368,24.422,154.087
C01330=1081.888,244.688,-80.380,175.371,24.426,154.087
C01331=1081.894,244.937,-80.407,175.373,24.429,154.088
C01332=1081.900,245.185,-80.435,175.376,24.432,154.088
C01333=1081.905,245.433,-80.462,175.378,24.435,154.089
C01334=1081.911,245.681,-80.489,175.381,24.439,154.089
C01335=1081.916,245.930,-80.516,175.383,24.442,154.089
C01336=1081.922,246.178,-80.543,175.386,24.445,154.090
C01337=1081.928,246.427,-80.569,175.389,24.448,154.090
C01338=1081.933,246.676,-80.597,175.392,24.452,154.091
C01339=1081.939,246.925,-80.624,175.394,24.455,154.091
C01340=1081.945,247.172,-80.651,175.397,24.459,154.091
C01341=1081.950,247.421,-80.678,175.399,24.462,154.092
C01342=1081.956,247.669,-80.705,175.402,24.465,154.092
C01343=1081.961,247.918,-80.732,175.404,24.469,154.093
C01344=1081.968,248.166,-80.760,175.407,24.472,154.093
C01345=1081.973,248.415,-80.787,175.409,24.475,154.093
C01346=1081.979,248.663,-80.814,175.411,24.479,154.094
C01347=1081.987,249.050,-80.857,175.416,24.484,154.094
C01348=1081.995,249.436,-80.898,175.419,24.489,154.095
C01349=1082.005,249.822,-80.941,175.424,24.495,154.096
C01350=1082.013,250.208,-80.983,175.428,24.500,154.096
C01351=1082.019,250.457,-81.011,175.431,24.503,154.097
C01352=1082.025,250.705,-81.038,175.433,24.506,154.097
C01353=1082.030,250.954,-81.066,175.436,24.510,154.097
C01354=1082.036,251.202,-81.092,175.438,24.513,154.098
C01355=1082.042,251.451,-81.120,175.441,24.517,154.098
C01356=1082.047,251.699,-81.147,175.443,24.520,154.099
C01357=1082.053,251.947,-81.175,175.446,24.523,154.099
C01358=1082.058,252.196,-81.202,175.448,24.527,154.099
C01359=1082.064,252.444,-81.230,175.451,24.530,154.100
C01360=1082.070,252.693,-81.257,175.454,24.533,154.100
C01361=1082.075,252.941,-81.284,175.457,24.537,154.101
C01362=1082.081,253.189,-81.312,175.459,24.540,154.101
C01363=1082.087,253.438,-81.340,175.462,24.544,154.102
C01364=1082.092,253.686,-81.367,175.464,24.547,154.102
C01365=1082.098,253.934,-81.395,175.467,24.550,154.102
C01366=1082.104,254.183,-81.422,175.470,24.554,154.103
C01367=1082.109,254.432,-81.450,175.472,24.557,154.103
C01368=1082.114,254.680,-81.477,175.475,24.560,154.103
C01369=1082.121,254.929,-81.505,175.477,24.564,154.104
C01370=1082.126,255.177,-81.533,175.480,24.567,154.104
C01371=1082.132,255.425,-81.560,175.482,24.570,154.105
C01372=1082.138,255.674,-81.588,175.486,24.574,154.105
C01373=1082.144,255.922,-81.616,175.488,24.577,154.105
C01374=1082.149,256.171,-81.643,175.491,24.581,154.106
C01375=1082.155,256.419,-81.671,175.493,24.584,154.106
C01376=1082.161,256.667,-81.699,175.496,24.587,154.107
C01377=1082.166,256.916,-81.726,175.498,24.590,154.107
C01378=1082.172,257.164,-81.754,175.501,24.594,154.107
C01379=1082.178,257.413,-81.782,175.504,24.598,154.108
C01380=1082.184,257.661,-81.810,175.506,24.601,154.108
C01381=1082.189,257.909,-81.837,175.509,24.604,154.109
C01382=1082.195,258.158,-81.865,175.511,24.607,154.109
C01383=1082.201,258.406,-81.893,175.515,24.611,154.109
C01384=1082.207,258.655,-81.921,175.517,24.614,154.110
C01385=1082.213,258.903,-81.949,175.520,24.618,154.110
C01386=1082.218,259.152,-81.976,175.523,24.621,154.111
C01387=1082.224,259.400,-82.003,175.525,24.624,154.111
C01388=1082.230,259.648,-82.032,175.528,24.628,154.111
C01389=1082.236,259.896,-82.060,175.530,24.631,154.112
C01390=1082.242,260.145,-82.088,175.533,24.635,154.112
C01391=1082.248,260.393,-82.115,175.535,24.638,154.113
C01392=1082.254,260.642,-82.144,175.538,24.641,154.113
C01393=1082.259,260.890,-82.172,175.541,24.645,154.113
C01394=1082.265,261.139,-82.200,175.544,24.648,154.114
C01395=1082.271,261.386,-82.227,175.547,24.652,154.114
C01396=1082.277,261.635,-82.256,175.549,24.655,154.115
C01397=1082.282,261.883,-82.284,175.552,24.658,154.115
C01398=1082.288,262.132,-82.312,175.554,24.661,154.115
C01399=1082.297,262.515,-82.355,175.559,24.666,154.116
C01400=1082.306,262.899,-82.398,175.563,24.672,154.117
C01401=1082.315,263.282,-82.441,175.567,24.677,154.117
C01402=1082.325,263.666,-82.485,175.571,24.682,154.118
C01403=1082.330,263.914,-82.512,175.574,24.685,154.118
C01404=1082.336,264.162,-82.542,175.577,24.689,154.119
C01405=1082.342,264.410,-82.569,175.579,24.692,154.119
C01406=1082.348,264.659,-82.598,175.582,24.696,154.119
C01407=1082.353,264.907,-82.626,175.585,24.699,154.120
C01408=1082.359,265.156,-82.654,175.587,24.702,154.120
C01409=1082.364,265.404,-82.682,175.590,24.706,154.121
C01410=1082.370,265.652,-82.711,175.592,24.709,154.121
C01411=1082.376,265.901,-82.739,175.595,24.712,154.121
C01412=1082.382,266.149,-82.767,175.598,24.716,154.122
C01413=1082.388,266.397,-82.796,175.600,24.720,154.122
C01414=1082.393,266.645,-82.824,175.603,24.723,154.123
C01415=1082.399,266.894,-82.853,175.606,24.726,154.123
C01416=1082.405,267.143,-82.882,175.609,24.730,154.124
C01417=1082.410,267.391,-82.910,175.612,24.733,154.124
C01418=1082.416,267.639,-82.939,175.614,24.736,154.124
C01419=1082.421,267.887,-82.967,175.617,24.740,154.125
C01420=1082.427,268.136,-82.995,175.620,24.744,154.125
C01421=1082.434,268.384,-83.024,175.622,24.747,154.126
C01422=1082.439,268.632,-83.052,175.625,24.751,154.126
C01423=1082.445,268.880,-83.081,175.627,24.754,154.127
C01424=1082.451,269.129,-83.109,175.630,24.757,154.127
C01425=1082.456,269.377,-83.138,175.633,24.761,154.127
C01426=1082.462,269.625,-83.167,175.636,24.764,154.128
C01427=1082.467,269.873,-83.195,175.639,24.768,154.128
C01428=1082.474,270.121,-83.224,175.642,24.771,154.128
C01429=1082.480,270.370,-83.252,175.644,24.775,154.129
C01430=1082.484,270.618,-83.281,175.647,24.778,154.129
C01431=1082.490,270.867,-83.310,175.650,24.782,154.130
C01432=1082.497,271.115,-83.339,175.652,24.785,154.130
C01433=1082.502,271.363,-83.367,175.655,24.788,154.131
C01434=1082.508,271.611,-83.396,175.658,24.792,154.131
C01435=1082.513,271.860,-83.425,175.660,24.796,154.132
C01436=1082.520,272.108,-83.454,175.663,24.799,154.132
C01437=1082.525,272.356,-83.482,175.665,24.802,154.132
C01438=1082.531,272.605,-83.511,175.669,24.806,154.133
C01439=1082.537,272.853,-83.540,175.672,24.809,154.133
C01440=1082.542,273.101,-83.568,175.674,24.812,154.134
C01441=1082.548,273.349,-83.597,175.677,24.816,154.134
C01442=1082.554,273.597,-83.627,175.680,24.820,154.135
C01443=1082.560,273.846,-83.655,175.682,24.823,154.135
C01444=1082.565,274.094,-83.684,175.685,24.827,154.135
C01445=1082.571,274.342,-83.714,175.688,24.830,154.136
C01446=1082.577,274.591,-83.742,175.690,24.834,154.136
C01447=1082.582,274.839,-83.771,175.693,24.837,154.137
C01448=1082.588,275.087,-83.800,175.696,24.841,154.137
C01449=1082.594,275.335,-83.829,175.698,24.844,154.137
C01450=1082.600,275.584,-83.858,175.701,24.848,154.138
C01451=1082.609,275.970,-83.904,175.706,24.853,154.139
C01452=1082.618,276.356,-83.949,175.710,24.859,154.139
C01453=1082.626,276.743,-83.994,175.714,24.864,154.140
C01454=1082.636,277.129,-84.039,175.719,24.870,154.141
C01455=1082.641,277.377,-84.069,175.722,24.873,154.141
C01456=1082.647,277.625,-84.098,175.724,24.877,154.142
C01457=1082.652,277.874,-84.127,175.727,24.880,154.142
C01458=1082.659,278.122,-84.156,175.730,24.884,154.142
C01459=1082.664,278.370,-84.186,175.733,24.887,154.143
C01460=1082.670,278.618,-84.215,175.735,24.891,154.143
C01461=1082.675,278.866,-84.244,175.738,24.894,154.144
C01462=1082.682,279.114,-84.273,175.741,24.898,154.144
C01463=1082.687,279.363,-84.303,175.743,24.902,154.145
C01464=1082.693,279.611,-84.332,175.746,24.905,154.145
C01465=1082.699,279.859,-84.362,175.749,24.909,154.145
C01466=1082.705,280.107,-84.391,175.752,24.912,154.146
C01467=1082.710,280.355,-84.420,175.755,24.916,154.146
C01468=1082.715,280.603,-84.450,175.758,24.919,154.147
C01469=1082.722,280.852,-84.479,175.761,24.923,154.147
C01470=1082.727,281.100,-84.508,175.763,24.926,154.148
C01471=1082.733,281.348,-84.537,175.766,24.930,154.148
C01472=1082.739,281.597,-84.567,175.769,24.933,154.148
C01473=1082.745,281.845,-84.597,175.771,24.937,154.149
C01474=1082.750,282.093,-84.626,175.774,24.940,154.149
C01475=1082.756,282.340,-84.656,175.777,24.944,154.150
C01476=1082.761,282.589,-84.685,175.780,24.948,154.150
C01477=1082.767,282.837,-84.715,175.782,24.951,154.151
C01478=1082.773,283.086,-84.745,175.785,24.955,154.151
C01479=1082.779,283.334,-84.774,175.788,24.959,154.152
C01480=1082.785,283.582,-84.804,175.791,24.963,154.152
C01481=1082.790,283.830,-84.834,175.793,24.966,154.153
C01482=1082.796,284.078,-84.863,175.796,24.969,154.153
C01483=1082.802,284.326,-84.893,175.799,24.973,154.154
C01484=1082.808,284.574,-84.923,175.803,24.977,154.154
C01485=1082.813,284.823,-84.952,175.805,24.980,154.155
C01486=1082.819,285.071,-84.982,175.808,24.984,154.155
C01487=1082.825,285.318,-85.011,175.811,24.988,154.155
C01488=1082.830,285.567,-85.041,175.814,24.991,154.156
C01489=1082.836,285.814,-85.071,175.816,24.994,154.156
C01490=1082.841,286.063,-85.101,175.819,24.998,154.157
C01491=1082.847,286.311,-85.131,175.822,25.002,154.157
C01492=1082.854,286.559,-85.160,175.825,25.006,154.158
C01493=1082.859,286.807,-85.190,175.827,25.009,154.158
C01494=1082.865,287.055,-85.220,175.830,25.012,154.159
C01495=1082.870,287.303,-85.250,175.833,25.016,154.159
C01496=1082.876,287.551,-85.280,175.836,25.020,154.159
C01497=1082.882,287.800,-85.310,175.838,25.024,154.160
C01498=1082.889,288.048,-85.340,175.841,25.027,154.160
C01499=1082.894,288.296,-85.370,175.844,25.031,154.161
C01500=1082.900,288.544,-85.400,175.847,25.035,154.161
C01501=1082.906,288.793,-85.430,175.850,25.038,154.162
C01502=1082.912,289.040,-85.460,175.853,25.042,154.162
C01503=1082.921,289.437,-85.507,175.857,25.047,154.163
C01504=1082.930,289.833,-85.555,175.862,25.053,154.164
C01505=1082.939,290.228,-85.604,175.866,25.059,154.164
C01506=1082.948,290.625,-85.651,175.871,25.065,154.165
C01507=1082.954,290.873,-85.682,175.874,25.069,154.166
C01508=1082.960,291.121,-85.712,175.877,25.073,154.166
C01509=1082.965,291.369,-85.742,175.880,25.076,154.167
C01510=1082.971,291.617,-85.772,175.883,25.080,154.167
C01511=1082.977,291.865,-85.802,175.885,25.084,154.168
C01512=1082.983,292.113,-85.833,175.888,25.087,154.168
C01513=1082.989,292.362,-85.863,175.891,25.091,154.169
C01514=1082.995,292.610,-85.893,175.894,25.095,154.169
C01515=1083.001,292.857,-85.923,175.897,25.099,154.170
C01516=1083.006,293.105,-85.954,175.899,25.102,154.170
C01517=1083.012,293.353,-85.985,175.902,25.106,154.170
C01518=1083.017,293.602,-86.014,175.905,25.110,154.171
C01519=1083.023,293.850,-86.045,175.908,25.113,154.171
C01520=1083.029,294.097,-86.075,175.911,25.117,154.172
C01521=1083.035,294.346,-86.106,175.913,25.120,154.172
C01522=1083.041,294.594,-86.136,175.916,25.124,154.173
C01523=1083.047,294.842,-86.167,175.919,25.128,154.173
C01524=1083.053,295.089,-86.197,175.922,25.132,154.174
C01525=1083.058,295.337,-86.228,175.925,25.136,154.174
C01526=1083.064,295.586,-86.259,175.928,25.140,154.175
C01527=1083.070,295.834,-86.289,175.930,25.143,154.175
C01528=1083.076,296.082,-86.319,175.933,25.147,154.176
C01529=1083.081,296.329,-86.350,175.936,25.151,154.176
C01530=1083.087,296.578,-86.381,175.939,25.154,154.177
C01531=1083.092,296.825,-86.411,175.942,25.158,154.177
C01532=1083.099,297.074,-86.442,175.945,25.162,154.178
C01533=1083.105,297.322,-86.472,175.949,25.165,154.178
C01534=1083.110,297.570,-86.503,175.951,25.169,154.179
C01535=1083.116,297.818,-86.533,175.954,25.173,154.179
C01536=1083.122,298.066,-86.564,175.957,25.177,154.180
C01537=1083.127,298.314,-86.595,175.960,25.180,154.180
C01538=1083.133,298.562,-86.625,175.963,25.184,154.181
C01539=1083.138,298.810,-86.657,175.966,25.188,154.181
C01540=1083.144,299.058,-86.687,175.968,25.192,154.182
C01541=1083.150,299.306,-86.719,175.971,25.196,154.182
C01542=1083.156,299.554,-86.749,175.974,25.200,154.183
C01543=1083.161,299.802,-86.780,175.977,25.204,154.183
C01544=1083.167,300.050,-86.811,175.980,25.208,154.184
C01545=1083.172,300.298,-86.842,175.983,25.212,154.184
C01546=1083.178,300.546,-86.873,175.986,25.215,154.185
C01547=1083.184,300.794,-86.904,175.989,25.219,154.185
C01548=1083.189,301.042,-86.935,175.991,25.223,154.186
C01549=1083.195,301.290,-86.966,175.994,25.227,154.186
C01550=1083.201,301.538,-86.996,175.997,25.231,154.187
C01551=1083.206,301.786,-87.028,176.000,25.235,154.187
C01552=1083.212,302.033,-87.058,176.003,25.239,154.188
C01553=1083.218,302.281,-87.090,176.006,25.243,154.189
C01554=1083.224,302.530,-87.121,176.009,25.247,154.189
C01555=1083.233,302.940,-87.172,176.013,25.253,154.190
C01556=1083.243,303.350,-87.224,176.018,25.259,154.191
C01557=1083.252,303.760,-87.275,176.023,25.266,154.192
C01558=1083.261,304.171,-87.327,176.028,25.273,154.193
C01559=1083.267,304.418,-87.358,176.030,25.276,154.193
C01560=1083.273,304.667,-87.389,176.033,25.280,154.194
C01561=1083.279,304.914,-87.421,176.036,25.284,154.194
C01562=1083.284,305.162,-87.451,176.039,25.288,154.195
C01563=1083.290,305.410,-87.483,176.042,25.291,154.195
C01564=1083.296,305.657,-87.514,176.045,25.295,154.196
C01565=1083.302,305.906,-87.545,176.048,25.299,154.196
C01566=1083.308,306.154,-87.577,176.051,25.303,154.197
C01567=1083.313,306.402,-87.607,176.054,25.307,154.197
C01568=1083.319,306.650,-87.639,176.057,25.311,154.198
C01569=1083.325,306.897,-87.670,176.060,25.315,154.198
C01570=1083.331,307.146,-87.702,176.063,25.319,154.199
C01571=1083.337,307.393,-87.733,176.066,25.323,154.199
C01572=1083.343,307.641,-87.765,176.069,25.327,154.200
C01573=1083.349,307.889,-87.797,176.071,25.331,154.200
C01574=1083.354,308.138,-87.828,176.074,25.335,154.201
C01575=1083.360,308.385,-87.859,176.077,25.338,154.202
C01576=1083.366,308.633,-87.891,176.080,25.342,154.202
C01577=1083.372,308.881,-87.923,176.083,25.346,154.203
C01578=1083.378,309.129,-87.953,176.086,25.350,154.203
C01579=1083.384,309.377,-87.985,176.089,25.354,154.204
C01580=1083.390,309.625,-88.017,176.092,25.358,154.204
C01581=1083.395,309.872,-88.049,176.095,25.362,154.205
C01582=1083.402,310.120,-88.080,176.098,25.367,154.205
C01583=1083.407,310.368,-88.112,176.101,25.371,154.206
C01584=1083.413,310.617,-88.143,176.104,25.374,154.206
C01585=1083.419,310.864,-88.174,176.107,25.378,154.207
C01586=1083.425,311.112,-88.206,176.110,25.382,154.207
C01587=1083.431,311.360,-88.238,176.113,25.386,154.208
C01588=1083.436,311.608,-88.270,176.116,25.390,154.209
C01589=1083.443,311.856,-88.301,176.119,25.394,154.209
C01590=1083.448,312.103,-88.333,176.122,25.398,154.210
C01591=1083.454,312.351,-88.365,176.125,25.402,154.210
C01592=1083.460,312.600,-88.397,176.128,25.406,154.211
C01593=1083.466,312.847,-88.428,176.131,25.410,154.211
C01594=1083.472,313.095,-88.460,176.134,25.414,154.212
C01595=1083.478,313.343,-88.492,176.137,25.418,154.212
C01596=1083.484,313.591,-88.524,176.140,25.422,154.213
C01597=1083.491,313.839,-88.555,176.143,25.426,154.213
C01598=1083.497,314.087,-88.587,176.146,25.430,154.214
C01599=1083.502,314.334,-88.619,176.149,25.434,154.215
C01600=1083.508,314.583,-88.651,176.152,25.438,154.215
C01601=1083.514,314.830,-88.684,176.154,25.442,154.216
C01602=1083.520,315.078,-88.716,176.157,25.446,154.216
C01603=1083.526,315.326,-88.747,176.160,25.450,154.217
C01604=1083.532,315.574,-88.779,176.163,25.454,154.217
C01605=1083.537,315.822,-88.811,176.166,25.458,154.218
C01606=1083.543,316.069,-88.844,176.169,25.463,154.219
C01607=1083.552,316.482,-88.898,176.174,25.470,154.220
C01608=1083.562,316.896,-88.951,176.179,25.477,154.221
C01609=1083.571,317.309,-89.005,176.184,25.483,154.222
C01610=1083.581,317.722,-89.059,176.189,25.490,154.223
C01611=1083.587,317.971,-89.091,176.192,25.495,154.223
C01612=1083.592,318.218,-89.124,176.195,25.499,154.224
C01613=1083.598,318.466,-89.156,176.198,25.503,154.224
C01614=1083.604,318.714,-89.188,176.201,25.507,154.225
C01615=1083.609,318.961,-89.220,176.204,25.511,154.226
C01616=1083.615,319.210,-89.253,176.207,25.516,154.226
C01617=1083.621,319.457,-89.286,176.210,25.520,154.227
C01618=1083.626,319.705,-89.317,176.212,25.524,154.227
C01619=1083.632,319.953,-89.349,176.215,25.528,154.228
C01620=1083.638,320.201,-89.383,176.218,25.532,154.229
C01621=1083.644,320.449,-89.415,176.221,25.536,154.229
C01622=1083.650,320.696,-89.447,176.224,25.541,154.230
C01623=1083.656,320.944,-89.479,176.227,25.545,154.231
C01624=1083.661,321.192,-89.512,176.231,25.550,154.231
C01625=1083.667,321.440,-89.545,176.234,25.554,154.232
C01626=1083.673,321.688,-89.577,176.237,25.558,154.232
C01627=1083.678,321.935,-89.610,176.240,25.562,154.233
C01628=1083.684,322.183,-89.642,176.243,25.567,154.234
C01629=1083.691,322.431,-89.675,176.246,25.571,154.234
C01630=1083.696,322.679,-89.708,176.249,25.575,154.235
C01631=1083.702,322.927,-89.740,176.252,25.579,154.235
C01632=1083.709,323.175,-89.773,176.255,25.583,154.236
C01633=1083.713,323.422,-89.806,176.258,25.588,154.237
C01634=1083.719,323.670,-89.838,176.261,25.592,154.237
C01635=1083.726,323.918,-89.871,176.264,25.596,154.238
C01636=1083.731,324.165,-89.904,176.266,25.600,154.238
C01637=1083.737,324.414,-89.936,176.269,25.605,154.239
C01638=1083.743,324.662,-89.969,176.272,25.609,154.240
C01639=1083.749,324.909,-90.002,176.276,25.614,154.240
C01640=1083.755,325.157,-90.035,176.279,25.618,154.241
C01641=1083.761,325.405,-90.068,176.282,25.622,154.242
C01642=1083.767,325.653,-90.100,176.285,25.626,154.242
C01643=1083.773,325.900,-90.133,176.288,25.631,154.243
C01644=1083.778,326.148,-90.166,176.291,25.635,154.244
C01645=1083.785,326.395,-90.199,176.294,25.639,154.244
C01646=1083.790,326.643,-90.232,176.297,25.644,154.245
C01647=1083.796,326.891,-90.265,176.300,25.648,154.245
C01648=1083.802,327.139,-90.298,176.303,25.652,154.246
C01649=1083.808,327.386,-90.331,176.306,25.657,154.247
C01650=1083.815,327.634,-90.364,176.309,25.661,154.247
C01651=1083.820,327.882,-90.397,176.312,25.665,154.248
C01652=1083.826,328.129,-90.430,176.315,25.670,154.249
C01653=1083.832,328.377,-90.463,176.318,25.674,154.249
C01654=1083.838,328.625,-90.496,176.321,25.678,154.250
C01655=1083.844,328.873,-90.529,176.324,25.683,154.251
C01656=1083.851,329.121,-90.562,176.327,25.687,154.251
C01657=1083.856,329.369,-90.596,176.331,25.691,154.252
C01658=1083.862,329.617,-90.628,176.334,25.696,154.252
C01659=1083.872,330.023,-90.683,176.338,25.703,154.254
C01660=1083.882,330.429,-90.737,176.343,25.710,154.255
C01661=1083.892,330.835,-90.791,176.349,25.717,154.256
C01662=1083.902,331.243,-90.847,176.354,25.725,154.257
C01663=1083.908,331.490,-90.879,176.357,25.729,154.257
C01664=1083.914,331.738,-90.913,176.360,25.733,154.258
C01665=1083.919,331.986,-90.946,176.363,25.738,154.259
C01666=1083.926,332.234,-90.979,176.366,25.743,154.259
C01667=1083.932,332.481,-91.013,176.369,25.747,154.260
C01668=1083.937,332.729,-91.046,176.372,25.752,154.261
C01669=1083.943,332.977,-91.079,176.375,25.756,154.261
C01670=1083.949,333.224,-91.113,176.378,25.761,154.262
C01671=1083.955,333.472,-91.146,176.381,25.765,154.263
C01672=1083.961,333.720,-91.180,176.385,25.770,154.264
C01673=1083.967,333.967,-91.214,176.388,25.775,154.264
C01674=1083.972,334.215,-91.247,176.390,25.779,154.265
C01675=1083.978,334.463,-91.281,176.393,25.783,154.266
C01676=1083.984,334.711,-91.315,176.396,25.788,154.266
C01677=1083.990,334.957,-91.348,176.399,25.793,154.267
C01678=1083.996,335.205,-91.381,176.403,25.797,154.268
C01679=1084.002,335.454,-91.415,176.406,25.802,154.268
C01680=1084.008,335.701,-91.449,176.409,25.807,154.269
C01681=1084.014,335.949,-91.483,176.412,25.811,154.270
C01682=1084.019,336.196,-91.517,176.416,25.816,154.270
C01683=1084.025,336.444,-91.551,176.418,25.821,154.271
C01684=1084.032,336.691,-91.583,176.421,25.825,154.272
C01685=1084.038,336.939,-91.618,176.424,25.830,154.273
C01686=1084.044,337.187,-91.651,176.427,25.834,154.273
C01687=1084.049,337.435,-91.685,176.431,25.839,154.274
C01688=1084.055,337.682,-91.719,176.434,25.844,154.275
C01689=1084.061,337.930,-91.753,176.437,25.848,154.275
C01690=1084.067,338.178,-91.787,176.440,25.852,154.276
C01691=1084.073,338.425,-91.821,176.443,25.858,154.277
C01692=1084.079,338.673,-91.854,176.446,25.863,154.278
C01693=1084.085,338.921,-91.889,176.449,25.867,154.278
C01694=1084.091,339.168,-91.923,176.452,25.872,154.279
C01695=1084.097,339.416,-91.956,176.456,25.876,154.280
C01696=1084.102,339.663,-91.990,176.459,25.881,154.281
C01697=1084.109,339.911,-92.025,176.461,25.886,154.281
C01698=1084.115,340.159,-92.059,176.464,25.891,154.282
C01699=1084.120,340.406,-92.093,176.468,25.896,154.283
C01700=1084.126,340.653,-92.127,176.471,25.900,154.284
C01701=1084.132,340.902,-92.161,176.474,25.905,154.284
C01702=1084.138,341.149,-92.195,176.477,25.910,154.285
C01703=1084.144,341.397,-92.229,176.480,25.915,154.286
C01704=1084.150,341.645,-92.264,176.483,25.919,154.287
C01705=1084.156,341.892,-92.298,176.486,25.924,154.287
C01706=1084.162,342.139,-92.332,176.489,25.929,154.288
C01707=1084.168,342.388,-92.367,176.493,25.934,154.289
C01708=1084.173,342.635,-92.401,176.496,25.939,154.290
C01709=1084.179,342.882,-92.435,176.499,25.944,154.290
C01710=1084.186,343.130,-92.469,176.502,25.949,154.291
C01711=1084.195,343.531,-92.524,176.507,25.957,154.292
C01712=1084.205,343.932,-92.580,176.512,25.964,154.294
C01713=1084.215,344.332,-92.636,176.517,25.972,154.295
C01714=1084.224,344.733,-92.692,176.522,25.980,154.296
C01715=1084.230,344.981,-92.726,176.526,25.985,154.297
C01716=1084.236,345.229,-92.761,176.528,25.990,154.298
C01717=1084.242,345.476,-92.795,176.531,25.995,154.298
C01718=1084.248,345.723,-92.830,176.535,26.000,154.299
C01719=1084.254,345.971,-92.865,176.538,26.005,154.300
C01720=1084.260,346.219,-92.899,176.541,26.010,154.301
C01721=1084.266,346.467,-92.933,176.544,26.015,154.302
C01722=1084.272,346.714,-92.969,176.547,26.020,154.302
C01723=1084.278,346.962,-93.003,176.550,26.024,154.303
C01724=1084.283,347.209,-93.038,176.554,26.030,154.304
C01725=1084.289,347.456,-93.072,176.557,26.034,154.305
C01726=1084.296,347.704,-93.107,176.560,26.039,154.306
C01727=1084.301,347.951,-93.142,176.563,26.045,154.306
C01728=1084.308,348.199,-93.177,176.566,26.050,154.307
C01729=1084.313,348.446,-93.211,176.569,26.055,154.308
C01730=1084.319,348.694,-93.246,176.573,26.060,154.309
C01731=1084.325,348.941,-93.281,176.576,26.065,154.310
C01732=1084.331,349.189,-93.315,176.579,26.070,154.311
C01733=1084.337,349.436,-93.350,176.582,26.075,154.311
C01734=1084.343,349.684,-93.385,176.585,26.080,154.312
C01735=1084.349,349.931,-93.420,176.589,26.085,154.313
C01736=1084.355,350.179,-93.455,176.591,26.090,154.314
C01737=1084.361,350.426,-93.490,176.594,26.095,154.315
C01738=1084.367,350.674,-93.525,176.598,26.100,154.315
C01739=1084.374,350.921,-93.560,176.601,26.106,154.316
C01740=1084.379,351.168,-93.595,176.605,26.111,154.317
C01741=1084.385,351.417,-93.630,176.607,26.116,154.318
C01742=1084.391,351.663,-93.665,176.610,26.121,154.319
C01743=1084.397,351.912,-93.700,176.614,26.126,154.320
C01744=1084.403,352.158,-93.735,176.617,26.131,154.321
C01745=1084.409,352.406,-93.771,176.620,26.137,154.321
C01746=1084.416,352.653,-93.806,176.623,26.142,154.322
C01747=1084.421,352.901,-93.840,176.626,26.147,154.323
C01748=1084.427,353.149,-93.876,176.630,26.152,154.324
C01749=1084.433,353.395,-93.911,176.633,26.157,154.325
C01750=1084.439,353.643,-93.947,176.636,26.163,154.326
C01751=1084.445,353.891,-93.982,176.639,26.168,154.327
C01752=1084.451,354.138,-94.016,176.642,26.173,154.327
C01753=1084.457,354.386,-94.052,176.646,26.179,154.328
C01754=1084.463,354.633,-94.088,176.648,26.184,154.329
C01755=1084.469,354.880,-94.123,176.652,26.189,154.330
C01756=1084.475,355.128,-94.158,176.655,26.194,154.331
C01757=1084.481,355.375,-94.194,176.659,26.200,154.332
C01758=1084.486,355.623,-94.229,176.661,26.205,154.333
C01759=1084.492,355.871,-94.264,176.665,26.210,154.334
C01760=1084.498,356.117,-94.299,176.668,26.216,154.335
C01761=1084.504,356.365,-94.335,176.671,26.221,154.335
C01762=1084.510,356.613,-94.371,176.674,26.227,154.336
C01763=1084.520,357.016,-94.429,176.679,26.235,154.338
C01764=1084.531,357.420,-94.487,176.684,26.244,154.339
C01765=1084.540,357.823,-94.545,176.690,26.253,154.341
C01766=1084.550,358.227,-94.603,176.695,26.262,154.342
C01767=1084.556,358.475,-94.639,176.699,26.267,154.343
C01768=1084.563,358.722,-94.674,176.702,26.273,154.344
C01769=1084.568,358.969,-94.710,176.705,26.278,154.345
C01770=1084.574,359.216,-94.746,176.708,26.283,154.346
C01771=1084.580,359.464,-94.781,176.712,26.289,154.347
C01772=1084.586,359.712,-94.817,176.715,26.294,154.348
C01773=1084.593,359.959,-94.854,176.718,26.300,154.349
C01774=1084.598,360.206,-94.889,176.721,26.306,154.350
C01775=1084.604,360.454,-94.925,176.725,26.311,154.351
C01776=1084.610,360.701,-94.960,176.727,26.317,154.351
C01777=1084.617,360.948,-94.997,176.731,26.323,154.353
C01778=1084.622,361.195,-95.032,176.734,26.328,154.353
C01779=1084.628,361.443,-95.068,176.737,26.334,154.354
C01780=1084.634,361.690,-95.104,176.740,26.339,154.355
C01781=1084.640,361.938,-95.140,176.744,26.345,154.356
C01782=1084.647,362.185,-95.177,176.747,26.350,154.357
C01783=1084.653,362.432,-95.212,176.750,26.356,154.358
C01784=1084.658,362.679,-95.248,176.753,26.362,154.359
C01785=1084.664,362.926,-95.284,176.757,26.367,154.360
C01786=1084.671,363.173,-95.321,176.759,26.373,154.361
C01787=1084.677,363.421,-95.356,176.763,26.379,154.362
C01788=1084.683,363.668,-95.393,176.766,26.384,154.363
C01789=1084.689,363.916,-95.428,176.769,26.390,154.364
C01790=1084.696,364.163,-95.465,176.772,26.395,154.365
C01791=1084.702,364.411,-95.501,176.776,26.401,154.366
C01792=1084.708,364.658,-95.537,176.779,26.407,154.367
C01793=1084.714,364.905,-95.574,176.782,26.413,154.368
C01794=1084.719,365.152,-95.609,176.786,26.419,154.369
C01795=1084.725,365.399,-95.646,176.789,26.424,154.370
C01796=1084.732,365.646,-95.682,176.792,26.430,154.371
C01797=1084.738,365.894,-95.718,176.795,26.436,154.372
C01798=1084.743,366.141,-95.755,176.798,26.442,154.373
C01799=1084.750,366.388,-95.792,176.802,26.448,154.374
C01800=1084.756,366.635,-95.828,176.805,26.453,154.375
C01801=1084.762,366.883,-95.865,176.809,26.459,154.376
C01802=1084.768,367.130,-95.901,176.811,26.465,154.377
C01803=1084.774,367.377,-95.937,176.815,26.471,154.378
C01804=1084.780,367.624,-95.974,176.818,26.477,154.379
C01805=1084.786,367.872,-96.011,176.821,26.483,154.380
C01806=1084.792,368.119,-96.047,176.825,26.489,154.381
C01807=1084.798,368.366,-96.084,176.827,26.495,154.382
C01808=1084.804,368.613,-96.121,176.831,26.501,154.383
C01809=1084.810,368.860,-96.157,176.835,26.507,154.384
C01810=1084.816,369.108,-96.194,176.837,26.513,154.386
C01811=1084.822,369.355,-96.231,176.841,26.519,154.387
C01812=1084.829,369.602,-96.267,176.844,26.525,154.388
C01813=1084.834,369.849,-96.304,176.847,26.531,154.389
C01814=1084.841,370.096,-96.340,176.851,26.537,154.390
C01815=1084.846,370.306,-96.372,176.854,26.542,154.391
C01816=1084.850,370.516,-96.402,176.857,26.547,154.392
C01817=1084.856,370.725,-96.434,176.859,26.552,154.392
C01818=1084.861,370.935,-96.465,176.862,26.558,154.393
